LIN {X 0,Y 389.55,Z 544.012,A -85,B 0,C 180,E1 -11990.321,E2 -11990.321} C_VEL
LIN {X 0,Y 389.974,Z 535.473,A -85,B 0,C 180,E1 -11990.85,E2 -11990.85} C_VEL
LIN {X 0,Y 386.923,Z 515.614,A -85,B 0,C 180,E1 -11992.126,E2 -11992.126} C_VEL
LIN {X 0,Y 383.966,Z 500.348,A -85,B 0,C 180,E1 -11992.925,E2 -11992.925} C_VEL
LIN {X 0,Y 382.611,Z 493.228,A -85,B 0,C 180,E1 -11993.24,E2 -11993.24} C_VEL
LIN {X 0,Y 382.976,Z 485.45,A -85,B 0,C 180,E1 -11996.718,E2 -11996.718} C_VEL
LIN {X 0,Y 383.373,Z 478.936,A -85,B 0,C 180,E1 -11999.667,E2 -11999.667} C_VEL
LIN {X 0,Y 383.827,Z 471.033,A -85,B 0,C 180,E1 -12003.32,E2 -12003.32} C_VEL
LIN {X 0,Y 384.194,Z 464.514,A -85,B 0,C 180,E1 -12006.401,E2 -12006.401} C_VEL
LIN {X 0,Y 384.639,Z 457.344,A -85,B 0,C 180,E1 -12009.878,E2 -12009.878} C_VEL
LIN {X 0,Y 385.108,Z 450.851,A -85,B 0,C 180,E1 -12013.116,E2 -12013.116} C_VEL
LIN {X 0,Y 385.546,Z 444.924,A -85,B 0,C 180,E1 -12016.157,E2 -12016.157} C_VEL
LIN {X 0,Y 385.519,Z 440.793,A -85,B 0,C 180,E1 -12018.368,E2 -12018.368} C_VEL
LIN {X 0,Y 384.796,Z 436.258,A -85,B 0,C 180,E1 -12020.941,E2 -12020.941} C_VEL
LIN {X 0,Y 383.623,Z 429.852,A -85,B 0,C 180,E1 -12024.754,E2 -12024.754} C_VEL
LIN {X 0,Y 383.043,Z 426.398,A -85,B 0,C 180,E1 -12027.007,E2 -12027.007} C_VEL
LIN {X 0,Y 382.993,Z 426.406,A -85,B 0,C 180,E1 -12030.3,E2 -12030.3} C_VEL
LIN {X 0,Y 383.058,Z 426.39,A -85,B 0,C 180,E1 -12032.698,E2 -12032.698} C_VEL
LIN {X 0,Y 383.054,Z 426.391,A -85,B 0,C 180,E1 -12035.04,E2 -12035.04} C_VEL
LIN {X 0,Y 382.995,Z 426.395,A -85,B 0,C 180,E1 -12038.469,E2 -12038.469} C_VEL
LIN {X 0,Y 383.091,Z 426.391,A -85,B 0,C 180,E1 -12041.828,E2 -12041.828} C_VEL
LIN {X 0,Y 383.112,Z 426.374,A -85,B 0,C 180,E1 -12045.118,E2 -12045.118} C_VEL
LIN {X 0,Y 383.099,Z 426.39,A -85,B 0,C 180,E1 -12048.358,E2 -12048.358} C_VEL
LIN {X 0,Y 383.23,Z 426.363,A -85,B 0,C 180,E1 -12052.013,E2 -12052.013} C_VEL
LIN {X 0,Y 383.199,Z 426.376,A -85,B 0,C 180,E1 -12054.739,E2 -12054.739} C_VEL
LIN {X 0,Y 383.387,Z 426.343,A -85,B 0,C 180,E1 -12057.899,E2 -12057.899} C_VEL
LIN {X 0,Y 383.522,Z 426.34,A -85,B 0,C 180,E1 -12060,E2 -12060} C_VEL
LIN {X 0,Y 383.248,Z 426.358,A -85,B 0,C 180,E1 -12063.154,E2 -12063.154} C_VEL
LIN {X 0,Y 383.271,Z 426.365,A -85,B 0,C 180,E1 -12066.637,E2 -12066.637} C_VEL
LIN {X 0,Y 383.262,Z 426.356,A -85,B 0,C 180,E1 -12068.436,E2 -12068.436} C_VEL
LIN {X 0,Y 383.1,Z 426.391,A -85,B 0,C 180,E1 -12071.642,E2 -12071.642} C_VEL
LIN {X 0,Y 383.112,Z 426.383,A -85,B 0,C 180,E1 -12074.882,E2 -12074.882} C_VEL
LIN {X 0,Y 383.065,Z 426.386,A -85,B 0,C 180,E1 -12078.174,E2 -12078.174} C_VEL
LIN {X 0,Y 382.994,Z 426.402,A -85,B 0,C 180,E1 -12081.531,E2 -12081.531} C_VEL
LIN {X 0,Y 383.052,Z 426.396,A -85,B 0,C 180,E1 -12084.96,E2 -12084.96} C_VEL
LIN {X 0,Y 383.042,Z 426.4,A -85,B 0,C 180,E1 -12088.493,E2 -12088.493} C_VEL
LIN {X 0,Y 383.011,Z 426.401,A -85,B 0,C 180,E1 -12092.15,E2 -12092.15} C_VEL
LIN {X 0,Y 383.019,Z 426.401,A -85,B 0,C 180,E1 -12094.668,E2 -12094.668} C_VEL
LIN {X 0,Y 383.001,Z 426.401,A -85,B 0,C 180,E1 -12097.904,E2 -12097.904} C_VEL
LIN {X 0,Y 382.987,Z 426.405,A -85,B 0,C 180,E1 -12101.347,E2 -12101.347} C_VEL
LIN {X 0,Y 383.037,Z 426.473,A -85,B 0,C 180,E1 -12104.763,E2 -12104.763} C_VEL
LIN {X 0,Y 384.737,Z 434.782,A -85,B 0,C 180,E1 -12107.861,E2 -12107.861} C_VEL
LIN {X 0,Y 385.867,Z 441.672,A -85,B 0,C 180,E1 -12110.396,E2 -12110.396} C_VEL
LIN {X 0,Y 385.944,Z 445.456,A -85,B 0,C 180,E1 -12111.747,E2 -12111.747} C_VEL
LIN {X 0,Y 385.278,Z 456.469,A -85,B 0,C 180,E1 -12115.564,E2 -12115.564} C_VEL
LIN {X 0,Y 384.788,Z 467.116,A -85,B 0,C 180,E1 -12119.242,E2 -12119.242} C_VEL
LIN {X 0,Y 384.378,Z 475.927,A -85,B 0,C 180,E1 -12122.209,E2 -12122.209} C_VEL
LIN {X 0,Y 383.988,Z 486.577,A -85,B 0,C 180,E1 -12125.681,E2 -12125.681} C_VEL
LIN {X 0,Y 383.851,Z 491.515,A -85,B 0,C 180,E1 -12127.165,E2 -12127.165} C_VEL
LIN {X 0,Y 387.586,Z 506.42,A -85,B 0,C 180,E1 -12127.781,E2 -12127.781} C_VEL
LIN {X 0,Y 390.26,Z 520.477,A -85,B 0,C 180,E1 -12128.521,E2 -12128.521} C_VEL
LIN {X 0,Y 390.956,Z 526.338,A -85,B 0,C 180,E1 -12128.872,E2 -12128.872} C_VEL
LIN {X 0,Y 390.117,Z 538.424,A -85,B 0,C 180,E1 -12129.602,E2 -12129.602} C_VEL
LIN {X 0,Y 388.997,Z 551.518,A -85,B 0,C 180,E1 -12130.611,E2 -12130.611} C_VEL
LIN {X 0,Y 387.734,Z 563.629,A -85,B 0,C 180,E1 -12131.78,E2 -12131.78} C_VEL
LIN {X 0,Y 386.48,Z 574.62,A -85,B 0,C 180,E1 -12133.085,E2 -12133.085} C_VEL
LIN {X 0,Y 385.225,Z 585.417,A -85,B 0,C 180,E1 -12134.661,E2 -12134.661} C_VEL
LIN {X 0,Y 384.25,Z 594.334,A -85,B 0,C 180,E1 -12136.245,E2 -12136.245} C_VEL
LIN {X 0,Y 383.456,Z 601.761,A -85,B 0,C 180,E1 -12137.832,E2 -12137.832} C_VEL
LIN {X 0,Y 382.777,Z 607.952,A -85,B 0,C 180,E1 -12139.42,E2 -12139.42} C_VEL
LIN {X 0,Y 382.143,Z 614.494,A -85,B 0,C 180,E1 -12141.539,E2 -12141.539} C_VEL
LIN {X 0,Y 381.849,Z 619.404,A -85,B 0,C 180,E1 -12143.66,E2 -12143.66} C_VEL
LIN {X 0,Y 381.636,Z 622.825,A -85,B 0,C 180,E1 -12145.776,E2 -12145.776} C_VEL
LIN {X 0,Y 381.552,Z 624.859,A -85,B 0,C 180,E1 -12147.889,E2 -12147.889} C_VEL
LIN {X 0,Y 381.572,Z 625.56,A -85,B 0,C 180,E1 -12150,E2 -12150} C_VEL
LIN {X 0,Y 381.551,Z 624.928,A -85,B 0,C 180,E1 -12152.111,E2 -12152.111} C_VEL
LIN {X 0,Y 381.634,Z 622.952,A -85,B 0,C 180,E1 -12154.224,E2 -12154.224} C_VEL
LIN {X 0,Y 381.808,Z 619.592,A -85,B 0,C 180,E1 -12156.341,E2 -12156.341} C_VEL
LIN {X 0,Y 382.137,Z 614.75,A -85,B 0,C 180,E1 -12158.461,E2 -12158.461} C_VEL
LIN {X 0,Y 382.73,Z 608.275,A -85,B 0,C 180,E1 -12160.581,E2 -12160.581} C_VEL
LIN {X 0,Y 383.546,Z 601.057,A -85,B 0,C 180,E1 -12162.433,E2 -12162.433} C_VEL
LIN {X 0,Y 384.407,Z 592.904,A -85,B 0,C 180,E1 -12164.134,E2 -12164.134} C_VEL
LIN {X 0,Y 385.575,Z 582.661,A -85,B 0,C 180,E1 -12165.867,E2 -12165.867} C_VEL
LIN {X 0,Y 386.791,Z 572.244,A -85,B 0,C 180,E1 -12167.31,E2 -12167.31} C_VEL
LIN {X 0,Y 387.323,Z 567.013,A -85,B 0,C 180,E1 -12167.939,E2 -12167.939} C_VEL
LIN {X 0,Y 387.168,Z 562.405,A -85,B 0,C 180,E1 -12168.481,E2 -12168.481} C_VEL
LIN {X 0,Y 385.32,Z 554.726,A -85,B 0,C 180,E1 -12169.375,E2 -12169.375} C_VEL
LIN {X 0,Y 383.5,Z 546.778,A -85,B 0,C 180,E1 -12170.208,E2 -12170.208} C_VEL
LIN {X 0,Y 383.264,Z 541.619,A -85,B 0,C 180,E1 -12170.642,E2 -12170.642} C_VEL
LIN {X 0,Y 384.198,Z 529.103,A -85,B 0,C 180,E1 -12171.46,E2 -12171.46} C_VEL
LIN {X 0,Y 384.104,Z 524.85,A -85,B 0,C 180,E1 -12171.709,E2 -12171.709} C_VEL
LIN {X 0,Y 381.821,Z 511.485,A -85,B 0,C 180,E1 -12172.486,E2 -12172.486} C_VEL
LIN {X 0,Y 378.417,Z 497.286,A -85,B 0,C 180,E1 -12173.156,E2 -12173.156} C_VEL
LIN {X 0,Y 376.897,Z 491.19,A -85,B 0,C 180,E1 -12173.417,E2 -12173.417} C_VEL
LIN {X 0,Y 377.325,Z 479.65,A -85,B 0,C 180,E1 -12177.15,E2 -12177.15} C_VEL
LIN {X 0,Y 377.798,Z 469.278,A -85,B 0,C 180,E1 -12180.663,E2 -12180.663} C_VEL
LIN {X 0,Y 378.339,Z 458.238,A -85,B 0,C 180,E1 -12184.511,E2 -12184.511} C_VEL
LIN {X 0,Y 379.011,Z 447.434,A -85,B 0,C 180,E1 -12188.303,E2 -12188.303} C_VEL
LIN {X 0,Y 379.019,Z 443.422,A -85,B 0,C 180,E1 -12189.754,E2 -12189.754} C_VEL
LIN {X 0,Y 378.012,Z 437.363,A -85,B 0,C 180,E1 -12192.014,E2 -12192.014} C_VEL
LIN {X 0,Y 376.299,Z 428.906,A -85,B 0,C 180,E1 -12195.212,E2 -12195.212} C_VEL
LIN {X 0,Y 375.959,Z 427.284,A -85,B 0,C 180,E1 -12195.836,E2 -12195.836} C_VEL
LIN {X 0,Y 375.942,Z 427.289,A -85,B 0,C 180,E1 -12199.133,E2 -12199.133} C_VEL
LIN {X 0,Y 375.967,Z 427.283,A -85,B 0,C 180,E1 -12201.912,E2 -12201.912} C_VEL
LIN {X 0,Y 375.982,Z 427.273,A -85,B 0,C 180,E1 -12205.333,E2 -12205.333} C_VEL
LIN {X 0,Y 375.962,Z 427.279,A -85,B 0,C 180,E1 -12208.438,E2 -12208.438} C_VEL
LIN {X 0,Y 376.004,Z 427.274,A -85,B 0,C 180,E1 -12212.142,E2 -12212.142} C_VEL
LIN {X 0,Y 376.023,Z 427.359,A -85,B 0,C 180,E1 -12215.39,E2 -12215.39} C_VEL
LIN {X 0,Y 381.008,Z 442.581,A -85,B 0,C 180,E1 -12216.589,E2 -12216.589} C_VEL
LIN {X 0,Y 384.181,Z 453.208,A -85,B 0,C 180,E1 -12217.55,E2 -12217.55} C_VEL
LIN {X 0,Y 382.956,Z 467.291,A -85,B 0,C 180,E1 -12218.749,E2 -12218.749} C_VEL
LIN {X 0,Y 381.648,Z 480.803,A -85,B 0,C 180,E1 -12220.158,E2 -12220.158} C_VEL
LIN {X 0,Y 380.365,Z 492.989,A -85,B 0,C 180,E1 -12221.693,E2 -12221.693} C_VEL
LIN {X 0,Y 379.267,Z 503.692,A -85,B 0,C 180,E1 -12223.308,E2 -12223.308} C_VEL
LIN {X 0,Y 378.205,Z 512.753,A -85,B 0,C 180,E1 -12224.921,E2 -12224.921} C_VEL
LIN {X 0,Y 377.419,Z 521.639,A -85,B 0,C 180,E1 -12226.814,E2 -12226.814} C_VEL
LIN {X 0,Y 376.623,Z 529.015,A -85,B 0,C 180,E1 -12228.7,E2 -12228.7} C_VEL
LIN {X 0,Y 376.043,Z 535.823,A -85,B 0,C 180,E1 -12230.859,E2 -12230.859} C_VEL
LIN {X 0,Y 375.611,Z 540.995,A -85,B 0,C 180,E1 -12232.948,E2 -12232.948} C_VEL
LIN {X 0,Y 375.491,Z 544.234,A -85,B 0,C 180,E1 -12234.63,E2 -12234.63} C_VEL
LIN {X 0,Y 375.294,Z 547.209,A -85,B 0,C 180,E1 -12236.779,E2 -12236.779} C_VEL
LIN {X 0,Y 374.988,Z 548.983,A -85,B 0,C 180,E1 -12238.926,E2 -12238.926} C_VEL
LIN {X 0,Y 375.03,Z 549.543,A -85,B 0,C 180,E1 -12241.074,E2 -12241.074} C_VEL
LIN {X 0,Y 375.315,Z 548.902,A -85,B 0,C 180,E1 -12243.22,E2 -12243.22} C_VEL
LIN {X 0,Y 375.838,Z 547.056,A -85,B 0,C 180,E1 -12245.365,E2 -12245.365} C_VEL
LIN {X 0,Y 376.224,Z 544.012,A -85,B 0,C 180,E1 -12247.514,E2 -12247.514} C_VEL
LIN {X 0,Y 376.901,Z 539.622,A -85,B 0,C 180,E1 -12249.661,E2 -12249.661} C_VEL
LIN {X 0,Y 377.559,Z 533.837,A -85,B 0,C 180,E1 -12251.815,E2 -12251.815} C_VEL
LIN {X 0,Y 378.769,Z 526.39,A -85,B 0,C 180,E1 -12253.958,E2 -12253.958} C_VEL
LIN {X 0,Y 379.802,Z 519.659,A -85,B 0,C 180,E1 -12255.554,E2 -12255.554} C_VEL
LIN {X 0,Y 381.234,Z 510.121,A -85,B 0,C 180,E1 -12257.432,E2 -12257.432} C_VEL
LIN {X 0,Y 382.539,Z 500.397,A -85,B 0,C 180,E1 -12259.032,E2 -12259.032} C_VEL
LIN {X 0,Y 384.197,Z 488.421,A -85,B 0,C 180,E1 -12260.65,E2 -12260.65} C_VEL
LIN {X 0,Y 385.845,Z 475.738,A -85,B 0,C 180,E1 -12262.066,E2 -12262.066} C_VEL
LIN {X 0,Y 387.215,Z 462.86,A -85,B 0,C 180,E1 -12263.251,E2 -12263.251} C_VEL
LIN {X 0,Y 387.867,Z 456.283,A -85,B 0,C 180,E1 -12263.77,E2 -12263.77} C_VEL
LIN {X 0,Y 384.824,Z 446.725,A -85,B 0,C 180,E1 -12264.838,E2 -12264.838} C_VEL
LIN {X 0,Y 379.638,Z 434.754,A -85,B 0,C 180,E1 -12266.212,E2 -12266.212} C_VEL
LIN {X 0,Y 376.181,Z 428.125,A -85,B 0,C 180,E1 -12267.01,E2 -12267.01} C_VEL
LIN {X 0,Y 376.012,Z 427.277,A -85,B 0,C 180,E1 -12267.125,E2 -12267.125} C_VEL
LIN {X 0,Y 375.957,Z 427.28,A -85,B 0,C 180,E1 -12270.694,E2 -12270.694} C_VEL
LIN {X 0,Y 375.961,Z 427.28,A -85,B 0,C 180,E1 -12274.111,E2 -12274.111} C_VEL
LIN {X 0,Y 375.954,Z 427.281,A -85,B 0,C 180,E1 -12276.741,E2 -12276.741} C_VEL
LIN {X 0,Y 375.972,Z 427.343,A -85,B 0,C 180,E1 -12279.137,E2 -12279.137} C_VEL
LIN {X 0,Y 376.756,Z 431.554,A -85,B 0,C 180,E1 -12282.186,E2 -12282.186} C_VEL
LIN {X 0,Y 377.08,Z 434.855,A -85,B 0,C 180,E1 -12284.228,E2 -12284.228} C_VEL
LIN {X 0,Y 376.323,Z 441.536,A -85,B 0,C 180,E1 -12287.754,E2 -12287.754} C_VEL
LIN {X 0,Y 376.101,Z 448.65,A -85,B 0,C 180,E1 -12291.186,E2 -12291.186} C_VEL
LIN {X 0,Y 375.976,Z 456.213,A -85,B 0,C 180,E1 -12294.586,E2 -12294.586} C_VEL
LIN {X 0,Y 375.765,Z 465.202,A -85,B 0,C 180,E1 -12298.42,E2 -12298.42} C_VEL
LIN {X 0,Y 375.648,Z 472.795,A -85,B 0,C 180,E1 -12301.561,E2 -12301.561} C_VEL
LIN {X 0,Y 375.447,Z 480.867,A -85,B 0,C 180,E1 -12304.812,E2 -12304.812} C_VEL
LIN {X 0,Y 376.282,Z 484.869,A -85,B 0,C 180,E1 -12305.069,E2 -12305.069} C_VEL
LIN {X 0,Y 378.786,Z 495.627,A -85,B 0,C 180,E1 -12305.81,E2 -12305.81} C_VEL
LIN {X 0,Y 380.799,Z 508.736,A -85,B 0,C 180,E1 -12306.713,E2 -12306.713} C_VEL
LIN {X 0,Y 381.881,Z 525.377,A -85,B 0,C 180,E1 -12307.924,E2 -12307.924} C_VEL
LIN {X 0,Y 382.948,Z 534.73,A -85,B 0,C 180,E1 -12308.699,E2 -12308.699} C_VEL
LIN {X 0,Y 383.303,Z 538.44,A -85,B 0,C 180,E1 -12308.952,E2 -12308.952} C_VEL
LIN {X 0,Y 382.313,Z 551.26,A -85,B 0,C 180,E1 -12309.83,E2 -12309.83} C_VEL
LIN {X 0,Y 381.121,Z 563.56,A -85,B 0,C 180,E1 -12310.894,E2 -12310.894} C_VEL
LIN {X 0,Y 379.885,Z 574.724,A -85,B 0,C 180,E1 -12312.087,E2 -12312.087} C_VEL
LIN {X 0,Y 378.643,Z 585.901,A -85,B 0,C 180,E1 -12313.557,E2 -12313.557} C_VEL
LIN {X 0,Y 377.481,Z 595.928,A -85,B 0,C 180,E1 -12315.174,E2 -12315.174} C_VEL
LIN {X 0,Y 376.63,Z 604.166,A -85,B 0,C 180,E1 -12316.786,E2 -12316.786} C_VEL
LIN {X 0,Y 375.739,Z 612.057,A -85,B 0,C 180,E1 -12318.674,E2 -12318.674} C_VEL
LIN {X 0,Y 375.247,Z 617.578,A -85,B 0,C 180,E1 -12320.296,E2 -12320.296} C_VEL
LIN {X 0,Y 374.792,Z 623.348,A -85,B 0,C 180,E1 -12322.457,E2 -12322.457} C_VEL
LIN {X 0,Y 374.702,Z 626.071,A -85,B 0,C 180,E1 -12323.763,E2 -12323.763} C_VEL
LIN {X 0,Y 374.607,Z 629.077,A -85,B 0,C 180,E1 -12325.696,E2 -12325.696} C_VEL
LIN {X 0,Y 374.53,Z 631.117,A -85,B 0,C 180,E1 -12327.849,E2 -12327.849} C_VEL
LIN {X 0,Y 374.546,Z 631.796,A -85,B 0,C 180,E1 -12330,E2 -12330} C_VEL
LIN {X 0,Y 374.53,Z 631.117,A -85,B 0,C 180,E1 -12332.151,E2 -12332.151} C_VEL
LIN {X 0,Y 374.594,Z 629.077,A -85,B 0,C 180,E1 -12334.304,E2 -12334.304} C_VEL
LIN {X 0,Y 374.681,Z 625.627,A -85,B 0,C 180,E1 -12336.462,E2 -12336.462} C_VEL
LIN {X 0,Y 374.978,Z 620.661,A -85,B 0,C 180,E1 -12338.623,E2 -12338.623} C_VEL
LIN {X 0,Y 375.515,Z 614.034,A -85,B 0,C 180,E1 -12340.787,E2 -12340.787} C_VEL
LIN {X 0,Y 376.348,Z 606.612,A -85,B 0,C 180,E1 -12342.675,E2 -12342.675} C_VEL
LIN {X 0,Y 377.09,Z 598.979,A -85,B 0,C 180,E1 -12344.269,E2 -12344.269} C_VEL
LIN {X 0,Y 378.186,Z 589.435,A -85,B 0,C 180,E1 -12345.909,E2 -12345.909} C_VEL
LIN {X 0,Y 379.33,Z 578.998,A -85,B 0,C 180,E1 -12347.383,E2 -12347.383} C_VEL
LIN {X 0,Y 380.726,Z 567.452,A -85,B 0,C 180,E1 -12348.707,E2 -12348.707} C_VEL
LIN {X 0,Y 381.944,Z 555.302,A -85,B 0,C 180,E1 -12349.84,E2 -12349.84} C_VEL
LIN {X 0,Y 383.036,Z 541.993,A -85,B 0,C 180,E1 -12350.823,E2 -12350.823} C_VEL
LIN {X 0,Y 383.234,Z 536.565,A -85,B 0,C 180,E1 -12351.164,E2 -12351.164} C_VEL
LIN {X 0,Y 380.34,Z 517.81,A -85,B 0,C 180,E1 -12352.353,E2 -12352.353} C_VEL
LIN {X 0,Y 377.516,Z 502.717,A -85,B 0,C 180,E1 -12353.202,E2 -12353.202} C_VEL
LIN {X 0,Y 375.59,Z 492.591,A -85,B 0,C 180,E1 -12353.661,E2 -12353.661} C_VEL
LIN {X 0,Y 375.896,Z 486.003,A -85,B 0,C 180,E1 -12356.662,E2 -12356.662} C_VEL
LIN {X 0,Y 376.368,Z 478.188,A -85,B 0,C 180,E1 -12360.277,E2 -12360.277} C_VEL
LIN {X 0,Y 376.896,Z 470.272,A -85,B 0,C 180,E1 -12364.015,E2 -12364.015} C_VEL
LIN {X 0,Y 377.333,Z 462.216,A -85,B 0,C 180,E1 -12367.926,E2 -12367.926} C_VEL
LIN {X 0,Y 377.797,Z 455.488,A -85,B 0,C 180,E1 -12371.283,E2 -12371.283} C_VEL
LIN {X 0,Y 378.387,Z 448.045,A -85,B 0,C 180,E1 -12375.106,E2 -12375.106} C_VEL
LIN {X 0,Y 378.569,Z 442.74,A -85,B 0,C 180,E1 -12377.952,E2 -12377.952} C_VEL
LIN {X 0,Y 377.865,Z 437.777,A -85,B 0,C 180,E1 -12380.775,E2 -12380.775} C_VEL
LIN {X 0,Y 376.678,Z 431.324,A -85,B 0,C 180,E1 -12384.662,E2 -12384.662} C_VEL
LIN {X 0,Y 375.994,Z 427.276,A -85,B 0,C 180,E1 -12387.26,E2 -12387.26} C_VEL
LIN {X 0,Y 375.972,Z 427.28,A -85,B 0,C 180,E1 -12390.921,E2 -12390.921} C_VEL
LIN {X 0,Y 376.007,Z 427.262,A -85,B 0,C 180,E1 -12394.539,E2 -12394.539} C_VEL
LIN {X 0,Y 375.965,Z 427.274,A -85,B 0,C 180,E1 -12398.046,E2 -12398.046} C_VEL
LIN {X 0,Y 376.026,Z 427.269,A -85,B 0,C 180,E1 -12401.474,E2 -12401.474} C_VEL
LIN {X 0,Y 376.06,Z 427.253,A -85,B 0,C 180,E1 -12404.833,E2 -12404.833} C_VEL
LIN {X 0,Y 376.052,Z 427.269,A -85,B 0,C 180,E1 -12408.137,E2 -12408.137} C_VEL
LIN {X 0,Y 376.202,Z 427.238,A -85,B 0,C 180,E1 -12411.938,E2 -12411.938} C_VEL
LIN {X 0,Y 376.171,Z 427.252,A -85,B 0,C 180,E1 -12414.64,E2 -12414.64} C_VEL
LIN {X 0,Y 376.354,Z 427.219,A -85,B 0,C 180,E1 -12417.86,E2 -12417.86} C_VEL
LIN {X 0,Y 376.491,Z 427.216,A -85,B 0,C 180,E1 -12420,E2 -12420} C_VEL
LIN {X 0,Y 376.186,Z 427.237,A -85,B 0,C 180,E1 -12423.213,E2 -12423.213} C_VEL
LIN {X 0,Y 376.236,Z 427.241,A -85,B 0,C 180,E1 -12426.628,E2 -12426.628} C_VEL
LIN {X 0,Y 376.207,Z 427.235,A -85,B 0,C 180,E1 -12428.595,E2 -12428.595} C_VEL
LIN {X 0,Y 376.053,Z 427.269,A -85,B 0,C 180,E1 -12431.863,E2 -12431.863} C_VEL
LIN {X 0,Y 376.06,Z 427.264,A -85,B 0,C 180,E1 -12435.167,E2 -12435.167} C_VEL
LIN {X 0,Y 376.011,Z 427.263,A -85,B 0,C 180,E1 -12438.527,E2 -12438.527} C_VEL
LIN {X 0,Y 375.959,Z 427.278,A -85,B 0,C 180,E1 -12441.955,E2 -12441.955} C_VEL
LIN {X 0,Y 376.007,Z 427.273,A -85,B 0,C 180,E1 -12445.461,E2 -12445.461} C_VEL
LIN {X 0,Y 375.972,Z 427.277,A -85,B 0,C 180,E1 -12449.079,E2 -12449.079} C_VEL
LIN {X 0,Y 375.951,Z 427.278,A -85,B 0,C 180,E1 -12452.829,E2 -12452.829} C_VEL
LIN {X 0,Y 375.959,Z 427.276,A -85,B 0,C 180,E1 -12455.416,E2 -12455.416} C_VEL
LIN {X 0,Y 375.976,Z 427.277,A -85,B 0,C 180,E1 -12458.271,E2 -12458.271} C_VEL
LIN {X 0,Y 375.937,Z 427.283,A -85,B 0,C 180,E1 -12461.601,E2 -12461.601} C_VEL
LIN {X 0,Y 375.97,Z 427.294,A -85,B 0,C 180,E1 -12464.288,E2 -12464.288} C_VEL
LIN {X 0,Y 377.584,Z 435.211,A -85,B 0,C 180,E1 -12467.289,E2 -12467.289} C_VEL
LIN {X 0,Y 378.728,Z 441.181,A -85,B 0,C 180,E1 -12469.538,E2 -12469.538} C_VEL
LIN {X 0,Y 379.072,Z 445.563,A -85,B 0,C 180,E1 -12471.14,E2 -12471.14} C_VEL
LIN {X 0,Y 378.42,Z 456.099,A -85,B 0,C 180,E1 -12474.849,E2 -12474.849} C_VEL
LIN {X 0,Y 377.901,Z 466.875,A -85,B 0,C 180,E1 -12478.619,E2 -12478.619} C_VEL
LIN {X 0,Y 377.485,Z 475.778,A -85,B 0,C 180,E1 -12481.656,E2 -12481.656} C_VEL
LIN {X 0,Y 377.031,Z 486.532,A -85,B 0,C 180,E1 -12485.203,E2 -12485.203} C_VEL
LIN {X 0,Y 376.905,Z 491.373,A -85,B 0,C 180,E1 -12486.718,E2 -12486.718} C_VEL
LIN {X 0,Y 380.862,Z 507.204,A -85,B 0,C 180,E1 -12487.394,E2 -12487.394} C_VEL
LIN {X 0,Y 383.401,Z 520.5,A -85,B 0,C 180,E1 -12488.117,E2 -12488.117} C_VEL
LIN {X 0,Y 384.26,Z 527.394,A -85,B 0,C 180,E1 -12488.543,E2 -12488.543} C_VEL
LIN {X 0,Y 383.316,Z 540.363,A -85,B 0,C 180,E1 -12489.362,E2 -12489.362} C_VEL
LIN {X 0,Y 382.167,Z 553.079,A -85,B 0,C 180,E1 -12490.39,E2 -12490.39} C_VEL
LIN {X 0,Y 380.84,Z 564.864,A -85,B 0,C 180,E1 -12491.577,E2 -12491.577} C_VEL
LIN {X 0,Y 379.65,Z 574.673,A -85,B 0,C 180,E1 -12492.771,E2 -12492.771} C_VEL
LIN {X 0,Y 378.365,Z 585.472,A -85,B 0,C 180,E1 -12494.375,E2 -12494.375} C_VEL
LIN {X 0,Y 377.28,Z 594.392,A -85,B 0,C 180,E1 -12495.986,E2 -12495.986} C_VEL
LIN {X 0,Y 376.506,Z 601.819,A -85,B 0,C 180,E1 -12497.604,E2 -12497.604} C_VEL
LIN {X 0,Y 375.762,Z 608.011,A -85,B 0,C 180,E1 -12499.22,E2 -12499.22} C_VEL
LIN {X 0,Y 375.105,Z 614.553,A -85,B 0,C 180,E1 -12501.38,E2 -12501.38} C_VEL
LIN {X 0,Y 374.781,Z 619.463,A -85,B 0,C 180,E1 -12503.54,E2 -12503.54} C_VEL
LIN {X 0,Y 374.566,Z 622.884,A -85,B 0,C 180,E1 -12505.696,E2 -12505.696} C_VEL
LIN {X 0,Y 374.45,Z 624.918,A -85,B 0,C 180,E1 -12507.849,E2 -12507.849} C_VEL
LIN {X 0,Y 374.473,Z 625.618,A -85,B 0,C 180,E1 -12510,E2 -12510} C_VEL
LIN {X 0,Y 374.449,Z 624.987,A -85,B 0,C 180,E1 -12512.151,E2 -12512.151} C_VEL
LIN {X 0,Y 374.564,Z 623.009,A -85,B 0,C 180,E1 -12514.304,E2 -12514.304} C_VEL
LIN {X 0,Y 374.724,Z 619.649,A -85,B 0,C 180,E1 -12516.461,E2 -12516.461} C_VEL
LIN {X 0,Y 375.099,Z 614.807,A -85,B 0,C 180,E1 -12518.621,E2 -12518.621} C_VEL
LIN {X 0,Y 375.7,Z 608.33,A -85,B 0,C 180,E1 -12520.782,E2 -12520.782} C_VEL
LIN {X 0,Y 376.578,Z 601.11,A -85,B 0,C 180,E1 -12522.667,E2 -12522.667} C_VEL
LIN {X 0,Y 377.43,Z 593.474,A -85,B 0,C 180,E1 -12524.296,E2 -12524.296} C_VEL
LIN {X 0,Y 378.52,Z 584.438,A -85,B 0,C 180,E1 -12525.894,E2 -12525.894} C_VEL
LIN {X 0,Y 379.742,Z 574.381,A -85,B 0,C 180,E1 -12527.363,E2 -12527.363} C_VEL
LIN {X 0,Y 381.052,Z 563.308,A -85,B 0,C 180,E1 -12528.691,E2 -12528.691} C_VEL
LIN {X 0,Y 382.373,Z 551.107,A -85,B 0,C 180,E1 -12529.879,E2 -12529.879} C_VEL
LIN {X 0,Y 383.264,Z 541.619,A -85,B 0,C 180,E1 -12530.642,E2 -12530.642} C_VEL
LIN {X 0,Y 382.939,Z 538.171,A -85,B 0,C 180,E1 -12530.927,E2 -12530.927} C_VEL
LIN {X 0,Y 380.764,Z 532.824,A -85,B 0,C 180,E1 -12531.426,E2 -12531.426} C_VEL
LIN {X 0,Y 377.761,Z 526.324,A -85,B 0,C 180,E1 -12532.01,E2 -12532.01} C_VEL
LIN {X 0,Y 377.167,Z 523.952,A -85,B 0,C 180,E1 -12532.182,E2 -12532.182} C_VEL
LIN {X 0,Y 374.655,Z 510.038,A -85,B 0,C 180,E1 -12533.002,E2 -12533.002} C_VEL
LIN {X 0,Y 371.097,Z 495.685,A -85,B 0,C 180,E1 -12533.677,E2 -12533.677} C_VEL
LIN {X 0,Y 369.974,Z 491.187,A -85,B 0,C 180,E1 -12533.882,E2 -12533.882} C_VEL
LIN {X 0,Y 370.444,Z 479.532,A -85,B 0,C 180,E1 -12537.698,E2 -12537.698} C_VEL
LIN {X 0,Y 370.892,Z 469.493,A -85,B 0,C 180,E1 -12541.143,E2 -12541.143} C_VEL
LIN {X 0,Y 371.429,Z 459.685,A -85,B 0,C 180,E1 -12544.586,E2 -12544.586} C_VEL
LIN {X 0,Y 372.137,Z 448.564,A -85,B 0,C 180,E1 -12548.552,E2 -12548.552} C_VEL
LIN {X 0,Y 372.076,Z 444.723,A -85,B 0,C 180,E1 -12549.957,E2 -12549.957} C_VEL
LIN {X 0,Y 371.004,Z 438.405,A -85,B 0,C 180,E1 -12552.372,E2 -12552.372} C_VEL
LIN {X 0,Y 369.5,Z 430.888,A -85,B 0,C 180,E1 -12555.271,E2 -12555.271} C_VEL
LIN {X 0,Y 368.887,Z 428.163,A -85,B 0,C 180,E1 -12556.383,E2 -12556.383} C_VEL
LIN {X 0,Y 368.914,Z 428.164,A -85,B 0,C 180,E1 -12559.643,E2 -12559.643} C_VEL
LIN {X 0,Y 368.904,Z 428.155,A -85,B 0,C 180,E1 -12563.144,E2 -12563.144} C_VEL
LIN {X 0,Y 368.898,Z 428.152,A -85,B 0,C 180,E1 -12566.462,E2 -12566.462} C_VEL
LIN {X 0,Y 368.925,Z 428.148,A -85,B 0,C 180,E1 -12570.31,E2 -12570.31} C_VEL
LIN {X 0,Y 368.984,Z 428.149,A -85,B 0,C 180,E1 -12573.535,E2 -12573.535} C_VEL
LIN {X 0,Y 368.995,Z 428.147,A -85,B 0,C 180,E1 -12575.02,E2 -12575.02} C_VEL
LIN {X 0,Y 374.008,Z 443.613,A -85,B 0,C 180,E1 -12576.277,E2 -12576.277} C_VEL
LIN {X 0,Y 377.363,Z 454.655,A -85,B 0,C 180,E1 -12577.31,E2 -12577.31} C_VEL
LIN {X 0,Y 376.135,Z 468.173,A -85,B 0,C 180,E1 -12578.488,E2 -12578.488} C_VEL
LIN {X 0,Y 374.899,Z 480.239,A -85,B 0,C 180,E1 -12579.755,E2 -12579.755} C_VEL
LIN {X 0,Y 373.552,Z 492.85,A -85,B 0,C 180,E1 -12581.347,E2 -12581.347} C_VEL
LIN {X 0,Y 372.42,Z 503.706,A -85,B 0,C 180,E1 -12582.992,E2 -12582.992} C_VEL
LIN {X 0,Y 371.328,Z 512.897,A -85,B 0,C 180,E1 -12584.635,E2 -12584.635} C_VEL
LIN {X 0,Y 370.487,Z 521.903,A -85,B 0,C 180,E1 -12586.563,E2 -12586.563} C_VEL
LIN {X 0,Y 369.65,Z 529.386,A -85,B 0,C 180,E1 -12588.484,E2 -12588.484} C_VEL
LIN {X 0,Y 369.047,Z 536.294,A -85,B 0,C 180,E1 -12590.684,E2 -12590.684} C_VEL
LIN {X 0,Y 368.577,Z 541.712,A -85,B 0,C 180,E1 -12592.888,E2 -12592.888} C_VEL
LIN {X 0,Y 368.437,Z 544.843,A -85,B 0,C 180,E1 -12594.527,E2 -12594.527} C_VEL
LIN {X 0,Y 368.259,Z 547.891,A -85,B 0,C 180,E1 -12596.718,E2 -12596.718} C_VEL
LIN {X 0,Y 367.937,Z 549.734,A -85,B 0,C 180,E1 -12598.905,E2 -12598.905} C_VEL
LIN {X 0,Y 367.98,Z 550.366,A -85,B 0,C 180,E1 -12601.094,E2 -12601.094} C_VEL
LIN {X 0,Y 368.284,Z 549.794,A -85,B 0,C 180,E1 -12603.282,E2 -12603.282} C_VEL
LIN {X 0,Y 368.831,Z 548.008,A -85,B 0,C 180,E1 -12605.467,E2 -12605.467} C_VEL
LIN {X 0,Y 369.263,Z 545.022,A -85,B 0,C 180,E1 -12607.656,E2 -12607.656} C_VEL
LIN {X 0,Y 369.977,Z 540.725,A -85,B 0,C 180,E1 -12609.844,E2 -12609.844} C_VEL
LIN {X 0,Y 370.707,Z 535.011,A -85,B 0,C 180,E1 -12612.037,E2 -12612.037} C_VEL
LIN {X 0,Y 371.986,Z 527.63,A -85,B 0,C 180,E1 -12614.218,E2 -12614.218} C_VEL
LIN {X 0,Y 373.133,Z 520.824,A -85,B 0,C 180,E1 -12615.882,E2 -12615.882} C_VEL
LIN {X 0,Y 374.626,Z 511.579,A -85,B 0,C 180,E1 -12617.749,E2 -12617.749} C_VEL
LIN {X 0,Y 376.005,Z 501.988,A -85,B 0,C 180,E1 -12619.376,E2 -12619.376} C_VEL
LIN {X 0,Y 377.598,Z 491.263,A -85,B 0,C 180,E1 -12620.893,E2 -12620.893} C_VEL
LIN {X 0,Y 379.358,Z 478.98,A -85,B 0,C 180,E1 -12622.32,E2 -12622.32} C_VEL
LIN {X 0,Y 380.796,Z 466.751,A -85,B 0,C 180,E1 -12623.523,E2 -12623.523} C_VEL
LIN {X 0,Y 381.671,Z 459.206,A -85,B 0,C 180,E1 -12624.147,E2 -12624.147} C_VEL
LIN {X 0,Y 380.728,Z 455.019,A -85,B 0,C 180,E1 -12624.615,E2 -12624.615} C_VEL
LIN {X 0,Y 376.706,Z 444.132,A -85,B 0,C 180,E1 -12625.927,E2 -12625.927} C_VEL
LIN {X 0,Y 370.633,Z 431.883,A -85,B 0,C 180,E1 -12627.497,E2 -12627.497} C_VEL
LIN {X 0,Y 369.191,Z 429.255,A -85,B 0,C 180,E1 -12627.847,E2 -12627.847} C_VEL
LIN {X 0,Y 368.968,Z 428.155,A -85,B 0,C 180,E1 -12627.97,E2 -12627.97} C_VEL
LIN {X 0,Y 368.911,Z 428.158,A -85,B 0,C 180,E1 -12630.987,E2 -12630.987} C_VEL
LIN {X 0,Y 368.937,Z 428.155,A -85,B 0,C 180,E1 -12634.853,E2 -12634.853} C_VEL
LIN {X 0,Y 368.949,Z 428.336,A -85,B 0,C 180,E1 -12638.648,E2 -12638.648} C_VEL
LIN {X 0,Y 369.71,Z 432.333,A -85,B 0,C 180,E1 -12641.708,E2 -12641.708} C_VEL
LIN {X 0,Y 370.099,Z 435.56,A -85,B 0,C 180,E1 -12643.813,E2 -12643.813} C_VEL
LIN {X 0,Y 369.586,Z 439.934,A -85,B 0,C 180,E1 -12646.27,E2 -12646.27} C_VEL
LIN {X 0,Y 369.12,Z 447.978,A -85,B 0,C 180,E1 -12650.369,E2 -12650.369} C_VEL
LIN {X 0,Y 368.97,Z 455.315,A -85,B 0,C 180,E1 -12653.809,E2 -12653.809} C_VEL
LIN {X 0,Y 368.773,Z 462.48,A -85,B 0,C 180,E1 -12656.987,E2 -12656.987} C_VEL
LIN {X 0,Y 368.625,Z 471.492,A -85,B 0,C 180,E1 -12660.84,E2 -12660.84} C_VEL
LIN {X 0,Y 368.391,Z 478.966,A -85,B 0,C 180,E1 -12663.953,E2 -12663.953} C_VEL
LIN {X 0,Y 369.157,Z 482.836,A -85,B 0,C 180,E1 -12664.219,E2 -12664.219} C_VEL
LIN {X 0,Y 369.913,Z 485.255,A -85,B 0,C 180,E1 -12664.416,E2 -12664.416} C_VEL
LIN {X 0,Y 372.772,Z 498.1,A -85,B 0,C 180,E1 -12665.377,E2 -12665.377} C_VEL
LIN {X 0,Y 374.515,Z 510.44,A -85,B 0,C 180,E1 -12666.291,E2 -12666.291} C_VEL
LIN {X 0,Y 375.305,Z 526.086,A -85,B 0,C 180,E1 -12667.509,E2 -12667.509} C_VEL
LIN {X 0,Y 376.255,Z 535.945,A -85,B 0,C 180,E1 -12668.381,E2 -12668.381} C_VEL
LIN {X 0,Y 376.602,Z 539.654,A -85,B 0,C 180,E1 -12668.638,E2 -12668.638} C_VEL
LIN {X 0,Y 375.479,Z 553.01,A -85,B 0,C 180,E1 -12669.595,E2 -12669.595} C_VEL
LIN {X 0,Y 374.263,Z 564.87,A -85,B 0,C 180,E1 -12670.673,E2 -12670.673} C_VEL
LIN {X 0,Y 372.858,Z 576.849,A -85,B 0,C 180,E1 -12672.022,E2 -12672.022} C_VEL
LIN {X 0,Y 371.592,Z 587.631,A -85,B 0,C 180,E1 -12673.519,E2 -12673.519} C_VEL
LIN {X 0,Y 370.419,Z 597.327,A -85,B 0,C 180,E1 -12675.16,E2 -12675.16} C_VEL
LIN {X 0,Y 369.53,Z 605.343,A -85,B 0,C 180,E1 -12676.807,E2 -12676.807} C_VEL
LIN {X 0,Y 368.723,Z 612.002,A -85,B 0,C 180,E1 -12678.455,E2 -12678.455} C_VEL
LIN {X 0,Y 368.199,Z 617.522,A -85,B 0,C 180,E1 -12680.108,E2 -12680.108} C_VEL
LIN {X 0,Y 367.829,Z 622.036,A -85,B 0,C 180,E1 -12681.761,E2 -12681.761} C_VEL
LIN {X 0,Y 367.593,Z 626.346,A -85,B 0,C 180,E1 -12683.82,E2 -12683.82} C_VEL
LIN {X 0,Y 367.51,Z 629.019,A -85,B 0,C 180,E1 -12685.613,E2 -12685.613} C_VEL
LIN {X 0,Y 367.427,Z 631.059,A -85,B 0,C 180,E1 -12687.808,E2 -12687.808} C_VEL
LIN {X 0,Y 367.446,Z 631.738,A -85,B 0,C 180,E1 -12690,E2 -12690} C_VEL
LIN {X 0,Y 367.427,Z 631.058,A -85,B 0,C 180,E1 -12692.192,E2 -12692.192} C_VEL
LIN {X 0,Y 367.496,Z 629.018,A -85,B 0,C 180,E1 -12694.387,E2 -12694.387} C_VEL
LIN {X 0,Y 367.595,Z 625.568,A -85,B 0,C 180,E1 -12696.587,E2 -12696.587} C_VEL
LIN {X 0,Y 367.944,Z 620.603,A -85,B 0,C 180,E1 -12698.79,E2 -12698.79} C_VEL
LIN {X 0,Y 368.495,Z 613.976,A -85,B 0,C 180,E1 -12700.995,E2 -12700.995} C_VEL
LIN {X 0,Y 369.382,Z 606.555,A -85,B 0,C 180,E1 -12702.918,E2 -12702.918} C_VEL
LIN {X 0,Y 370.161,Z 598.923,A -85,B 0,C 180,E1 -12704.542,E2 -12704.542} C_VEL
LIN {X 0,Y 371.341,Z 589.381,A -85,B 0,C 180,E1 -12706.21,E2 -12706.21} C_VEL
LIN {X 0,Y 372.555,Z 578.946,A -85,B 0,C 180,E1 -12707.709,E2 -12707.709} C_VEL
LIN {X 0,Y 373.993,Z 567.403,A -85,B 0,C 180,E1 -12709.057,E2 -12709.057} C_VEL
LIN {X 0,Y 375.302,Z 554.7,A -85,B 0,C 180,E1 -12710.257,E2 -12710.257} C_VEL
LIN {X 0,Y 376.392,Z 541.947,A -85,B 0,C 180,E1 -12711.209,E2 -12711.209} C_VEL
LIN {X 0,Y 376.509,Z 537.649,A -85,B 0,C 180,E1 -12711.489,E2 -12711.489} C_VEL
LIN {X 0,Y 374.588,Z 524.889,A -85,B 0,C 180,E1 -12712.324,E2 -12712.324} C_VEL
LIN {X 0,Y 370.506,Z 502.226,A -85,B 0,C 180,E1 -12713.618,E2 -12713.618} C_VEL
LIN {X 0,Y 368.538,Z 491.907,A -85,B 0,C 180,E1 -12714.106,E2 -12714.106} C_VEL
LIN {X 0,Y 368.867,Z 485.24,A -85,B 0,C 180,E1 -12717.211,E2 -12717.211} C_VEL
LIN {X 0,Y 369.296,Z 478.733,A -85,B 0,C 180,E1 -12720.286,E2 -12720.286} C_VEL
LIN {X 0,Y 369.831,Z 470.814,A -85,B 0,C 180,E1 -12724.097,E2 -12724.097} C_VEL
LIN {X 0,Y 370.313,Z 462.747,A -85,B 0,C 180,E1 -12728.083,E2 -12728.083} C_VEL
LIN {X 0,Y 370.804,Z 455.911,A -85,B 0,C 180,E1 -12731.557,E2 -12731.557} C_VEL
LIN {X 0,Y 371.341,Z 449.292,A -85,B 0,C 180,E1 -12735.011,E2 -12735.011} C_VEL
LIN {X 0,Y 371.587,Z 444.664,A -85,B 0,C 180,E1 -12737.53,E2 -12737.53} C_VEL
LIN {X 0,Y 371.129,Z 440.461,A -85,B 0,C 180,E1 -12739.92,E2 -12739.92} C_VEL
LIN {X 0,Y 370.219,Z 435.542,A -85,B 0,C 180,E1 -12742.873,E2 -12742.873} C_VEL
LIN {X 0,Y 369.118,Z 429.112,A -85,B 0,C 180,E1 -12746.904,E2 -12746.904} C_VEL
LIN {X 0,Y 368.926,Z 428.157,A -85,B 0,C 180,E1 -12747.546,E2 -12747.546} C_VEL
LIN {X 0,Y 368.981,Z 428.15,A -85,B 0,C 180,E1 -12751.564,E2 -12751.564} C_VEL
LIN {X 0,Y 369.001,Z 428.132,A -85,B 0,C 180,E1 -12754.02,E2 -12754.02} C_VEL
LIN {X 0,Y 368.934,Z 428.151,A -85,B 0,C 180,E1 -12757.605,E2 -12757.605} C_VEL
LIN {X 0,Y 368.984,Z 428.146,A -85,B 0,C 180,E1 -12761.107,E2 -12761.107} C_VEL
LIN {X 0,Y 368.999,Z 428.134,A -85,B 0,C 180,E1 -12764.535,E2 -12764.535} C_VEL
LIN {X 0,Y 369.007,Z 428.147,A -85,B 0,C 180,E1 -12767.907,E2 -12767.907} C_VEL
LIN {X 0,Y 369.149,Z 428.116,A -85,B 0,C 180,E1 -12771.889,E2 -12771.889} C_VEL
LIN {X 0,Y 369.143,Z 428.128,A -85,B 0,C 180,E1 -12774.538,E2 -12774.538} C_VEL
LIN {X 0,Y 369.319,Z 428.095,A -85,B 0,C 180,E1 -12777.819,E2 -12777.819} C_VEL
LIN {X 0,Y 369.46,Z 428.091,A -85,B 0,C 180,E1 -12780,E2 -12780} C_VEL
LIN {X 0,Y 369.318,Z 428.096,A -85,B 0,C 180,E1 -12782.181,E2 -12782.181} C_VEL
LIN {X 0,Y 369.206,Z 428.118,A -85,B 0,C 180,E1 -12786.615,E2 -12786.615} C_VEL
LIN {X 0,Y 369.139,Z 428.115,A -85,B 0,C 180,E1 -12788.761,E2 -12788.761} C_VEL
LIN {X 0,Y 369.008,Z 428.144,A -85,B 0,C 180,E1 -12792.093,E2 -12792.093} C_VEL
LIN {X 0,Y 369,Z 428.147,A -85,B 0,C 180,E1 -12795.465,E2 -12795.465} C_VEL
LIN {X 0,Y 368.96,Z 428.141,A -85,B 0,C 180,E1 -12798.894,E2 -12798.894} C_VEL
LIN {X 0,Y 368.926,Z 428.149,A -85,B 0,C 180,E1 -12802.396,E2 -12802.396} C_VEL
LIN {X 0,Y 369.001,Z 428.142,A -85,B 0,C 180,E1 -12805.98,E2 -12805.98} C_VEL
LIN {X 0,Y 368.963,Z 428.151,A -85,B 0,C 180,E1 -12808.812,E2 -12808.812} C_VEL
LIN {X 0,Y 368.9,Z 428.158,A -85,B 0,C 180,E1 -12812.238,E2 -12812.238} C_VEL
LIN {X 0,Y 368.93,Z 428.154,A -85,B 0,C 180,E1 -12815.002,E2 -12815.002} C_VEL
LIN {X 0,Y 368.911,Z 428.159,A -85,B 0,C 180,E1 -12818.64,E2 -12818.64} C_VEL
LIN {X 0,Y 368.883,Z 428.163,A -85,B 0,C 180,E1 -12822.01,E2 -12822.01} C_VEL
LIN {X 0,Y 368.931,Z 428.292,A -85,B 0,C 180,E1 -12823.843,E2 -12823.843} C_VEL
LIN {X 0,Y 370.584,Z 436.288,A -85,B 0,C 180,E1 -12826.943,E2 -12826.943} C_VEL
LIN {X 0,Y 371.91,Z 443.229,A -85,B 0,C 180,E1 -12829.596,E2 -12829.596} C_VEL
LIN {X 0,Y 372.162,Z 448.257,A -85,B 0,C 180,E1 -12831.451,E2 -12831.451} C_VEL
LIN {X 0,Y 371.428,Z 459.4,A -85,B 0,C 180,E1 -12835.414,E2 -12835.414} C_VEL
LIN {X 0,Y 370.905,Z 470.242,A -85,B 0,C 180,E1 -12839.229,E2 -12839.229} C_VEL
LIN {X 0,Y 370.448,Z 479.225,A -85,B 0,C 180,E1 -12842.302,E2 -12842.302} C_VEL
LIN {X 0,Y 369.992,Z 491.399,A -85,B 0,C 180,E1 -12846.258,E2 -12846.258} C_VEL
LIN {X 0,Y 373.906,Z 506.919,A -85,B 0,C 180,E1 -12846.939,E2 -12846.939} C_VEL
LIN {X 0,Y 376.625,Z 520.589,A -85,B 0,C 180,E1 -12847.705,E2 -12847.705} C_VEL
LIN {X 0,Y 377.58,Z 528.532,A -85,B 0,C 180,E1 -12848.209,E2 -12848.209} C_VEL
LIN {X 0,Y 376.551,Z 542.04,A -85,B 0,C 180,E1 -12849.104,E2 -12849.104} C_VEL
LIN {X 0,Y 375.329,Z 554.521,A -85,B 0,C 180,E1 -12850.16,E2 -12850.16} C_VEL
LIN {X 0,Y 373.894,Z 566.064,A -85,B 0,C 180,E1 -12851.365,E2 -12851.365} C_VEL
LIN {X 0,Y 372.637,Z 576.645,A -85,B 0,C 180,E1 -12852.72,E2 -12852.72} C_VEL
LIN {X 0,Y 371.305,Z 587.126,A -85,B 0,C 180,E1 -12854.352,E2 -12854.352} C_VEL
LIN {X 0,Y 370.321,Z 594.449,A -85,B 0,C 180,E1 -12855.717,E2 -12855.717} C_VEL
LIN {X 0,Y 369.556,Z 601.877,A -85,B 0,C 180,E1 -12857.367,E2 -12857.367} C_VEL
LIN {X 0,Y 368.733,Z 608.069,A -85,B 0,C 180,E1 -12859.012,E2 -12859.012} C_VEL
LIN {X 0,Y 368.055,Z 614.612,A -85,B 0,C 180,E1 -12861.213,E2 -12861.213} C_VEL
LIN {X 0,Y 367.695,Z 619.522,A -85,B 0,C 180,E1 -12863.415,E2 -12863.415} C_VEL
LIN {X 0,Y 367.475,Z 622.943,A -85,B 0,C 180,E1 -12865.613,E2 -12865.613} C_VEL
LIN {X 0,Y 367.352,Z 624.977,A -85,B 0,C 180,E1 -12867.807,E2 -12867.807} C_VEL
LIN {X 0,Y 367.373,Z 625.677,A -85,B 0,C 180,E1 -12870,E2 -12870} C_VEL
LIN {X 0,Y 367.351,Z 625.045,A -85,B 0,C 180,E1 -12872.193,E2 -12872.193} C_VEL
LIN {X 0,Y 367.473,Z 623.067,A -85,B 0,C 180,E1 -12874.387,E2 -12874.387} C_VEL
LIN {X 0,Y 367.647,Z 619.706,A -85,B 0,C 180,E1 -12876.586,E2 -12876.586} C_VEL
LIN {X 0,Y 368.048,Z 614.863,A -85,B 0,C 180,E1 -12878.787,E2 -12878.787} C_VEL
LIN {X 0,Y 368.503,Z 610.169,A -85,B 0,C 180,E1 -12880.439,E2 -12880.439} C_VEL
LIN {X 0,Y 369.346,Z 603.363,A -85,B 0,C 180,E1 -12882.361,E2 -12882.361} C_VEL
LIN {X 0,Y 370.205,Z 596.25,A -85,B 0,C 180,E1 -12884.007,E2 -12884.007} C_VEL
LIN {X 0,Y 371.268,Z 587.688,A -85,B 0,C 180,E1 -12885.649,E2 -12885.649} C_VEL
LIN {X 0,Y 372.563,Z 577.317,A -85,B 0,C 180,E1 -12887.284,E2 -12887.284} C_VEL
LIN {X 0,Y 374.008,Z 565.718,A -85,B 0,C 180,E1 -12888.772,E2 -12888.772} C_VEL
LIN {X 0,Y 375.374,Z 554.097,A -85,B 0,C 180,E1 -12889.98,E2 -12889.98} C_VEL
LIN {X 0,Y 376.617,Z 541.651,A -85,B 0,C 180,E1 -12891.025,E2 -12891.025} C_VEL
LIN {X 0,Y 377.646,Z 527.781,A -85,B 0,C 180,E1 -12891.932,E2 -12891.932} C_VEL
LIN {X 0,Y 377.167,Z 523.952,A -85,B 0,C 180,E1 -12892.182,E2 -12892.182} C_VEL
LIN {X 0,Y 375.653,Z 518.798,A -85,B 0,C 180,E1 -12892.557,E2 -12892.557} C_VEL
LIN {X 0,Y 371.309,Z 510.894,A -85,B 0,C 180,E1 -12893.194,E2 -12893.194} C_VEL
LIN {X 0,Y 366.698,Z 502.905,A -85,B 0,C 180,E1 -12893.783,E2 -12893.783} C_VEL
LIN {X 0,Y 364.72,Z 497.606,A -85,B 0,C 180,E1 -12894.067,E2 -12894.067} C_VEL
LIN {X 0,Y 363.033,Z 491.182,A -85,B 0,C 180,E1 -12894.368,E2 -12894.368} C_VEL
LIN {X 0,Y 363.47,Z 481.27,A -85,B 0,C 180,E1 -12897.649,E2 -12897.649} C_VEL
LIN {X 0,Y 363.938,Z 472.157,A -85,B 0,C 180,E1 -12900.78,E2 -12900.78} C_VEL
LIN {X 0,Y 364.523,Z 461.203,A -85,B 0,C 180,E1 -12904.664,E2 -12904.664} C_VEL
LIN {X 0,Y 365.268,Z 450.024,A -85,B 0,C 180,E1 -12908.706,E2 -12908.706} C_VEL
LIN {X 0,Y 365.167,Z 445.985,A -85,B 0,C 180,E1 -12910.207,E2 -12910.207} C_VEL
LIN {X 0,Y 363.984,Z 439.297,A -85,B 0,C 180,E1 -12912.8,E2 -12912.8} C_VEL
LIN {X 0,Y 362.414,Z 431.522,A -85,B 0,C 180,E1 -12915.849,E2 -12915.849} C_VEL
LIN {X 0,Y 361.843,Z 429.043,A -85,B 0,C 180,E1 -12916.91,E2 -12916.91} C_VEL
LIN {X 0,Y 361.857,Z 429.039,A -85,B 0,C 180,E1 -12920.139,E2 -12920.139} C_VEL
LIN {X 0,Y 361.87,Z 429.031,A -85,B 0,C 180,E1 -12922.982,E2 -12922.982} C_VEL
LIN {X 0,Y 361.86,Z 429.029,A -85,B 0,C 180,E1 -12926.63,E2 -12926.63} C_VEL
LIN {X 0,Y 361.878,Z 429.022,A -85,B 0,C 180,E1 -12929.672,E2 -12929.672} C_VEL
LIN {X 0,Y 361.957,Z 429.024,A -85,B 0,C 180,E1 -12933.475,E2 -12933.475} C_VEL
LIN {X 0,Y 361.937,Z 429.025,A -85,B 0,C 180,E1 -12934.672,E2 -12934.672} C_VEL
LIN {X 0,Y 366.535,Z 443.053,A -85,B 0,C 180,E1 -12935.821,E2 -12935.821} C_VEL
LIN {X 0,Y 370.358,Z 455.4,A -85,B 0,C 180,E1 -12936.992,E2 -12936.992} C_VEL
LIN {X 0,Y 369.994,Z 461.948,A -85,B 0,C 180,E1 -12937.555,E2 -12937.555} C_VEL
LIN {X 0,Y 368.617,Z 475.572,A -85,B 0,C 180,E1 -12938.886,E2 -12938.886} C_VEL
LIN {X 0,Y 367.235,Z 488.586,A -85,B 0,C 180,E1 -12940.433,E2 -12940.433} C_VEL
LIN {X 0,Y 365.956,Z 500.266,A -85,B 0,C 180,E1 -12942.105,E2 -12942.105} C_VEL
LIN {X 0,Y 364.821,Z 510.092,A -85,B 0,C 180,E1 -12943.78,E2 -12943.78} C_VEL
LIN {X 0,Y 363.875,Z 518.449,A -85,B 0,C 180,E1 -12945.458,E2 -12945.458} C_VEL
LIN {X 0,Y 362.985,Z 526.656,A -85,B 0,C 180,E1 -12947.419,E2 -12947.419} C_VEL
LIN {X 0,Y 362.318,Z 533.448,A -85,B 0,C 180,E1 -12949.381,E2 -12949.381} C_VEL
LIN {X 0,Y 361.759,Z 539.671,A -85,B 0,C 180,E1 -12951.622,E2 -12951.622} C_VEL
LIN {X 0,Y 361.38,Z 544.457,A -85,B 0,C 180,E1 -12953.86,E2 -12953.86} C_VEL
LIN {X 0,Y 361.325,Z 547.144,A -85,B 0,C 180,E1 -12955.538,E2 -12955.538} C_VEL
LIN {X 0,Y 361.01,Z 549.672,A -85,B 0,C 180,E1 -12957.769,E2 -12957.769} C_VEL
LIN {X 0,Y 360.878,Z 550.989,A -85,B 0,C 180,E1 -12960,E2 -12960} C_VEL
LIN {X 0,Y 361.059,Z 551.093,A -85,B 0,C 180,E1 -12962.231,E2 -12962.231} C_VEL
LIN {X 0,Y 361.554,Z 549.981,A -85,B 0,C 180,E1 -12964.459,E2 -12964.459} C_VEL
LIN {X 0,Y 361.968,Z 547.699,A -85,B 0,C 180,E1 -12966.69,E2 -12966.69} C_VEL
LIN {X 0,Y 362.644,Z 544.136,A -85,B 0,C 180,E1 -12968.919,E2 -12968.919} C_VEL
LIN {X 0,Y 363.464,Z 539.2,A -85,B 0,C 180,E1 -12971.149,E2 -12971.149} C_VEL
LIN {X 0,Y 364.202,Z 534.54,A -85,B 0,C 180,E1 -12972.821,E2 -12972.821} C_VEL
LIN {X 0,Y 365.402,Z 527.921,A -85,B 0,C 180,E1 -12974.764,E2 -12974.764} C_VEL
LIN {X 0,Y 366.669,Z 520.906,A -85,B 0,C 180,E1 -12976.466,E2 -12976.466} C_VEL
LIN {X 0,Y 368.262,Z 511.626,A -85,B 0,C 180,E1 -12978.354,E2 -12978.354} C_VEL
LIN {X 0,Y 369.838,Z 501.877,A -85,B 0,C 180,E1 -12980.002,E2 -12980.002} C_VEL
LIN {X 0,Y 371.721,Z 489.749,A -85,B 0,C 180,E1 -12981.702,E2 -12981.702} C_VEL
LIN {X 0,Y 373.565,Z 477.358,A -85,B 0,C 180,E1 -12983.124,E2 -12983.124} C_VEL
LIN {X 0,Y 375.318,Z 463.305,A -85,B 0,C 180,E1 -12984.455,E2 -12984.455} C_VEL
LIN {X 0,Y 375.375,Z 459.945,A -85,B 0,C 180,E1 -12984.764,E2 -12984.764} C_VEL
LIN {X 0,Y 371.779,Z 449.338,A -85,B 0,C 180,E1 -12986.112,E2 -12986.112} C_VEL
LIN {X 0,Y 366.412,Z 437.765,A -85,B 0,C 180,E1 -12987.685,E2 -12987.685} C_VEL
LIN {X 0,Y 362.127,Z 430.076,A -85,B 0,C 180,E1 -12988.816,E2 -12988.816} C_VEL
LIN {X 0,Y 361.926,Z 429.031,A -85,B 0,C 180,E1 -12988.932,E2 -12988.932} C_VEL
LIN {X 0,Y 361.849,Z 429.038,A -85,B 0,C 180,E1 -12992.945,E2 -12992.945} C_VEL
LIN {X 0,Y 361.869,Z 429.036,A -85,B 0,C 180,E1 -12995.637,E2 -12995.637} C_VEL
LIN {X 0,Y 361.882,Z 429.123,A -85,B 0,C 180,E1 -12997.933,E2 -12997.933} C_VEL
LIN {X 0,Y 362.623,Z 433.165,A -85,B 0,C 180,E1 -13001.22,E2 -13001.22} C_VEL
LIN {X 0,Y 363.097,Z 436.33,A -85,B 0,C 180,E1 -13003.403,E2 -13003.403} C_VEL
LIN {X 0,Y 362.925,Z 439.018,A -85,B 0,C 180,E1 -13005.023,E2 -13005.023} C_VEL
LIN {X 0,Y 362.218,Z 446.69,A -85,B 0,C 180,E1 -13009.174,E2 -13009.174} C_VEL
LIN {X 0,Y 361.942,Z 454.464,A -85,B 0,C 180,E1 -13012.991,E2 -13012.991} C_VEL
LIN {X 0,Y 361.757,Z 461.506,A -85,B 0,C 180,E1 -13016.236,E2 -13016.236} C_VEL
LIN {X 0,Y 361.502,Z 469.202,A -85,B 0,C 180,E1 -13019.637,E2 -13019.637} C_VEL
LIN {X 0,Y 361.42,Z 475.093,A -85,B 0,C 180,E1 -13022.18,E2 -13022.18} C_VEL
LIN {X 0,Y 361.39,Z 476.997,A -85,B 0,C 180,E1 -13022.995,E2 -13022.995} C_VEL
LIN {X 0,Y 362.206,Z 481.102,A -85,B 0,C 180,E1 -13023.314,E2 -13023.314} C_VEL
LIN {X 0,Y 362.942,Z 483.295,A -85,B 0,C 180,E1 -13023.518,E2 -13023.518} C_VEL
LIN {X 0,Y 365.891,Z 495.497,A -85,B 0,C 180,E1 -13024.525,E2 -13024.525} C_VEL
LIN {X 0,Y 367.995,Z 509.479,A -85,B 0,C 180,E1 -13025.64,E2 -13025.64} C_VEL
LIN {X 0,Y 368.754,Z 524.46,A -85,B 0,C 180,E1 -13026.864,E2 -13026.864} C_VEL
LIN {X 0,Y 369.24,Z 534.243,A -85,B 0,C 180,E1 -13027.772,E2 -13027.772} C_VEL
LIN {X 0,Y 369.96,Z 539.968,A -85,B 0,C 180,E1 -13028.258,E2 -13028.258} C_VEL
LIN {X 0,Y 368.798,Z 553.08,A -85,B 0,C 180,E1 -13029.218,E2 -13029.218} C_VEL
LIN {X 0,Y 367.535,Z 564.829,A -85,B 0,C 180,E1 -13030.304,E2 -13030.304} C_VEL
LIN {X 0,Y 366.087,Z 576.803,A -85,B 0,C 180,E1 -13031.678,E2 -13031.678} C_VEL
LIN {X 0,Y 364.739,Z 587.582,A -85,B 0,C 180,E1 -13033.2,E2 -13033.2} C_VEL
LIN {X 0,Y 363.51,Z 597.275,A -85,B 0,C 180,E1 -13034.871,E2 -13034.871} C_VEL
LIN {X 0,Y 362.558,Z 605.289,A -85,B 0,C 180,E1 -13036.549,E2 -13036.549} C_VEL
LIN {X 0,Y 361.739,Z 611.947,A -85,B 0,C 180,E1 -13038.229,E2 -13038.229} C_VEL
LIN {X 0,Y 361.168,Z 617.466,A -85,B 0,C 180,E1 -13039.914,E2 -13039.914} C_VEL
LIN {X 0,Y 360.663,Z 623.234,A -85,B 0,C 180,E1 -13042.16,E2 -13042.16} C_VEL
LIN {X 0,Y 360.446,Z 627.419,A -85,B 0,C 180,E1 -13044.405,E2 -13044.405} C_VEL
LIN {X 0,Y 360.337,Z 630.152,A -85,B 0,C 180,E1 -13046.646,E2 -13046.646} C_VEL
LIN {X 0,Y 360.344,Z 631.51,A -85,B 0,C 180,E1 -13048.882,E2 -13048.882} C_VEL
LIN {X 0,Y 360.344,Z 631.509,A -85,B 0,C 180,E1 -13051.118,E2 -13051.118} C_VEL
LIN {X 0,Y 360.335,Z 630.151,A -85,B 0,C 180,E1 -13053.354,E2 -13053.354} C_VEL
LIN {X 0,Y 360.413,Z 627.416,A -85,B 0,C 180,E1 -13055.595,E2 -13055.595} C_VEL
LIN {X 0,Y 360.659,Z 623.224,A -85,B 0,C 180,E1 -13057.84,E2 -13057.84} C_VEL
LIN {X 0,Y 361.149,Z 617.451,A -85,B 0,C 180,E1 -13060.087,E2 -13060.087} C_VEL
LIN {X 0,Y 361.887,Z 610.924,A -85,B 0,C 180,E1 -13062.05,E2 -13062.05} C_VEL
LIN {X 0,Y 362.751,Z 603.099,A -85,B 0,C 180,E1 -13063.947,E2 -13063.947} C_VEL
LIN {X 0,Y 363.86,Z 594.254,A -85,B 0,C 180,E1 -13065.689,E2 -13065.689} C_VEL
LIN {X 0,Y 365.126,Z 583.877,A -85,B 0,C 180,E1 -13067.358,E2 -13067.358} C_VEL
LIN {X 0,Y 366.446,Z 573.416,A -85,B 0,C 180,E1 -13068.738,E2 -13068.738} C_VEL
LIN {X 0,Y 367.859,Z 562.005,A -85,B 0,C 180,E1 -13069.969,E2 -13069.969} C_VEL
LIN {X 0,Y 369.049,Z 550.031,A -85,B 0,C 180,E1 -13071.019,E2 -13071.019} C_VEL
LIN {X 0,Y 369.964,Z 539.863,A -85,B 0,C 180,E1 -13071.742,E2 -13071.742} C_VEL
LIN {X 0,Y 368.116,Z 527.06,A -85,B 0,C 180,E1 -13072.631,E2 -13072.631} C_VEL
LIN {X 0,Y 365.597,Z 512.743,A -85,B 0,C 180,E1 -13073.421,E2 -13073.421} C_VEL
LIN {X 0,Y 362.461,Z 496.362,A -85,B 0,C 180,E1 -13074.312,E2 -13074.312} C_VEL
LIN {X 0,Y 361.482,Z 491.236,A -85,B 0,C 180,E1 -13074.55,E2 -13074.55} C_VEL
LIN {X 0,Y 361.853,Z 484.452,A -85,B 0,C 180,E1 -13077.784,E2 -13077.784} C_VEL
LIN {X 0,Y 362.28,Z 478.097,A -85,B 0,C 180,E1 -13080.854,E2 -13080.854} C_VEL
LIN {X 0,Y 362.785,Z 471.317,A -85,B 0,C 180,E1 -13084.18,E2 -13084.18} C_VEL
LIN {X 0,Y 363.277,Z 463.244,A -85,B 0,C 180,E1 -13088.249,E2 -13088.249} C_VEL
LIN {X 0,Y 363.791,Z 456.376,A -85,B 0,C 180,E1 -13091.797,E2 -13091.797} C_VEL
LIN {X 0,Y 364.398,Z 449.407,A -85,B 0,C 180,E1 -13095.529,E2 -13095.529} C_VEL
LIN {X 0,Y 364.586,Z 445.689,A -85,B 0,C 180,E1 -13097.57,E2 -13097.57} C_VEL
LIN {X 0,Y 363.97,Z 440.825,A -85,B 0,C 180,E1 -13100.416,E2 -13100.416} C_VEL
LIN {X 0,Y 362.961,Z 435.281,A -85,B 0,C 180,E1 -13103.803,E2 -13103.803} C_VEL
LIN {X 0,Y 362.108,Z 430.186,A -85,B 0,C 180,E1 -13107.082,E2 -13107.082} C_VEL
LIN {X 0,Y 361.879,Z 429.035,A -85,B 0,C 180,E1 -13107.883,E2 -13107.883} C_VEL
LIN {X 0,Y 361.901,Z 429.033,A -85,B 0,C 180,E1 -13110.955,E2 -13110.955} C_VEL
LIN {X 0,Y 361.956,Z 429.01,A -85,B 0,C 180,E1 -13113.475,E2 -13113.475} C_VEL
LIN {X 0,Y 361.892,Z 429.033,A -85,B 0,C 180,E1 -13117.145,E2 -13117.145} C_VEL
LIN {X 0,Y 361.922,Z 429.021,A -85,B 0,C 180,E1 -13120.724,E2 -13120.724} C_VEL
LIN {X 0,Y 361.947,Z 429.015,A -85,B 0,C 180,E1 -13124.226,E2 -13124.226} C_VEL
LIN {X 0,Y 362,Z 429.01,A -85,B 0,C 180,E1 -13126.528,E2 -13126.528} C_VEL
LIN {X 0,Y 362.002,Z 429.009,A -85,B 0,C 180,E1 -13129.937,E2 -13129.937} C_VEL
LIN {X 0,Y 362.153,Z 428.997,A -85,B 0,C 180,E1 -13133.314,E2 -13133.314} C_VEL
LIN {X 0,Y 362.283,Z 428.97,A -85,B 0,C 180,E1 -13137.777,E2 -13137.777} C_VEL
LIN {X 0,Y 362.43,Z 428.967,A -85,B 0,C 180,E1 -13140,E2 -13140} C_VEL
LIN {X 0,Y 362.282,Z 428.972,A -85,B 0,C 180,E1 -13142.224,E2 -13142.224} C_VEL
LIN {X 0,Y 362.174,Z 428.995,A -85,B 0,C 180,E1 -13146.686,E2 -13146.686} C_VEL
LIN {X 0,Y 362.076,Z 428.995,A -85,B 0,C 180,E1 -13148.933,E2 -13148.933} C_VEL
LIN {X 0,Y 361.962,Z 429.02,A -85,B 0,C 180,E1 -13152.332,E2 -13152.332} C_VEL
LIN {X 0,Y 361.964,Z 429.015,A -85,B 0,C 180,E1 -13154.62,E2 -13154.62} C_VEL
LIN {X 0,Y 361.958,Z 429.015,A -85,B 0,C 180,E1 -13158.1,E2 -13158.1} C_VEL
LIN {X 0,Y 361.863,Z 429.034,A -85,B 0,C 180,E1 -13161.655,E2 -13161.655} C_VEL
LIN {X 0,Y 361.929,Z 429.029,A -85,B 0,C 180,E1 -13165.29,E2 -13165.29} C_VEL
LIN {X 0,Y 361.92,Z 429.028,A -85,B 0,C 180,E1 -13167.778,E2 -13167.778} C_VEL
LIN {X 0,Y 361.848,Z 429.038,A -85,B 0,C 180,E1 -13171.285,E2 -13171.285} C_VEL
LIN {X 0,Y 361.856,Z 429.037,A -85,B 0,C 180,E1 -13174.28,E2 -13174.28} C_VEL
LIN {X 0,Y 361.865,Z 429.036,A -85,B 0,C 180,E1 -13177.223,E2 -13177.223} C_VEL
LIN {X 0,Y 361.838,Z 429.043,A -85,B 0,C 180,E1 -13180.756,E2 -13180.756} C_VEL
LIN {X 0,Y 361.864,Z 429.202,A -85,B 0,C 180,E1 -13183.341,E2 -13183.341} C_VEL
LIN {X 0,Y 363.596,Z 437.073,A -85,B 0,C 180,E1 -13186.455,E2 -13186.455} C_VEL
LIN {X 0,Y 364.862,Z 443.842,A -85,B 0,C 180,E1 -13189.087,E2 -13189.087} C_VEL
LIN {X 0,Y 365.296,Z 447.755,A -85,B 0,C 180,E1 -13190.588,E2 -13190.588} C_VEL
LIN {X 0,Y 364.838,Z 455.349,A -85,B 0,C 180,E1 -13193.333,E2 -13193.333} C_VEL
LIN {X 0,Y 364.303,Z 464.631,A -85,B 0,C 180,E1 -13196.663,E2 -13196.663} C_VEL
LIN {X 0,Y 363.805,Z 475.192,A -85,B 0,C 180,E1 -13200.379,E2 -13200.379} C_VEL
LIN {X 0,Y 363.216,Z 486.456,A -85,B 0,C 180,E1 -13204.192,E2 -13204.192} C_VEL
LIN {X 0,Y 363.08,Z 491.488,A -85,B 0,C 180,E1 -13205.78,E2 -13205.78} C_VEL
LIN {X 0,Y 367.071,Z 506.932,A -85,B 0,C 180,E1 -13206.485,E2 -13206.485} C_VEL
LIN {X 0,Y 369.825,Z 520.83,A -85,B 0,C 180,E1 -13207.283,E2 -13207.283} C_VEL
LIN {X 0,Y 370.912,Z 529.711,A -85,B 0,C 180,E1 -13207.871,E2 -13207.871} C_VEL
LIN {X 0,Y 369.835,Z 542.941,A -85,B 0,C 180,E1 -13208.779,E2 -13208.779} C_VEL
LIN {X 0,Y 368.472,Z 555.959,A -85,B 0,C 180,E1 -13209.921,E2 -13209.921} C_VEL
LIN {X 0,Y 367.01,Z 567.263,A -85,B 0,C 180,E1 -13211.147,E2 -13211.147} C_VEL
LIN {X 0,Y 365.594,Z 578.613,A -85,B 0,C 180,E1 -13212.665,E2 -13212.665} C_VEL
LIN {X 0,Y 364.223,Z 588.777,A -85,B 0,C 180,E1 -13214.327,E2 -13214.327} C_VEL
LIN {X 0,Y 363.304,Z 595.837,A -85,B 0,C 180,E1 -13215.721,E2 -13215.721} C_VEL
LIN {X 0,Y 362.446,Z 603.034,A -85,B 0,C 180,E1 -13217.4,E2 -13217.4} C_VEL
LIN {X 0,Y 361.538,Z 609.91,A -85,B 0,C 180,E1 -13219.358,E2 -13219.358} C_VEL
LIN {X 0,Y 360.887,Z 616.075,A -85,B 0,C 180,E1 -13221.602,E2 -13221.602} C_VEL
LIN {X 0,Y 360.611,Z 620.341,A -85,B 0,C 180,E1 -13223.694,E2 -13223.694} C_VEL
LIN {X 0,Y 360.389,Z 623.002,A -85,B 0,C 180,E1 -13225.526,E2 -13225.526} C_VEL
LIN {X 0,Y 360.257,Z 625.036,A -85,B 0,C 180,E1 -13227.764,E2 -13227.764} C_VEL
LIN {X 0,Y 360.274,Z 625.735,A -85,B 0,C 180,E1 -13230,E2 -13230} C_VEL
LIN {X 0,Y 360.256,Z 625.103,A -85,B 0,C 180,E1 -13232.236,E2 -13232.236} C_VEL
LIN {X 0,Y 360.385,Z 623.124,A -85,B 0,C 180,E1 -13234.474,E2 -13234.474} C_VEL
LIN {X 0,Y 360.582,Z 619.763,A -85,B 0,C 180,E1 -13236.716,E2 -13236.716} C_VEL
LIN {X 0,Y 361.018,Z 614.919,A -85,B 0,C 180,E1 -13238.96,E2 -13238.96} C_VEL
LIN {X 0,Y 361.667,Z 608.441,A -85,B 0,C 180,E1 -13241.205,E2 -13241.205} C_VEL
LIN {X 0,Y 362.703,Z 601.217,A -85,B 0,C 180,E1 -13243.16,E2 -13243.16} C_VEL
LIN {X 0,Y 363.671,Z 593.215,A -85,B 0,C 180,E1 -13244.926,E2 -13244.926} C_VEL
LIN {X 0,Y 365.063,Z 582.806,A -85,B 0,C 180,E1 -13246.784,E2 -13246.784} C_VEL
LIN {X 0,Y 366.415,Z 572.379,A -85,B 0,C 180,E1 -13248.305,E2 -13248.305} C_VEL
LIN {X 0,Y 367.888,Z 560.867,A -85,B 0,C 180,E1 -13249.676,E2 -13249.676} C_VEL
LIN {X 0,Y 369.345,Z 548.099,A -85,B 0,C 180,E1 -13250.903,E2 -13250.903} C_VEL
LIN {X 0,Y 370.604,Z 534.518,A -85,B 0,C 180,E1 -13251.927,E2 -13251.927} C_VEL
LIN {X 0,Y 370.887,Z 527.922,A -85,B 0,C 180,E1 -13252.345,E2 -13252.345} C_VEL
LIN {X 0,Y 368.785,Z 514.853,A -85,B 0,C 180,E1 -13253.181,E2 -13253.181} C_VEL
LIN {X 0,Y 365.537,Z 500.572,A -85,B 0,C 180,E1 -13253.928,E2 -13253.928} C_VEL
LIN {X 0,Y 364.72,Z 497.606,A -85,B 0,C 180,E1 -13254.067,E2 -13254.067} C_VEL
LIN {X 0,Y 363.623,Z 494.401,A -85,B 0,C 180,E1 -13254.317,E2 -13254.317} C_VEL
LIN {X 0,Y 361.941,Z 491.236,A -85,B 0,C 180,E1 -13254.808,E2 -13254.808} C_VEL
LIN {X 0,Y 359.59,Z 487.988,A -85,B 0,C 180,E1 -13255.68,E2 -13255.68} C_VEL
LIN {X 0,Y 357.377,Z 484.892,A -85,B 0,C 180,E1 -13256.882,E2 -13256.882} C_VEL
LIN {X 0,Y 356.598,Z 482.381,A -85,B 0,C 180,E1 -13257.812,E2 -13257.812} C_VEL
LIN {X 0,Y 356.574,Z 481.492,A -85,B 0,C 180,E1 -13258.122,E2 -13258.122} C_VEL
LIN {X 0,Y 357.075,Z 471.952,A -85,B 0,C 180,E1 -13261.438,E2 -13261.438} C_VEL
LIN {X 0,Y 357.623,Z 462.747,A -85,B 0,C 180,E1 -13264.744,E2 -13264.744} C_VEL
LIN {X 0,Y 358.411,Z 451.483,A -85,B 0,C 180,E1 -13268.865,E2 -13268.865} C_VEL
LIN {X 0,Y 358.278,Z 447.557,A -85,B 0,C 180,E1 -13270.341,E2 -13270.341} C_VEL
LIN {X 0,Y 356.832,Z 439.387,A -85,B 0,C 180,E1 -13273.578,E2 -13273.578} C_VEL
LIN {X 0,Y 355.146,Z 431.567,A -85,B 0,C 180,E1 -13276.722,E2 -13276.722} C_VEL
LIN {X 0,Y 354.791,Z 429.925,A -85,B 0,C 180,E1 -13277.446,E2 -13277.446} C_VEL
LIN {X 0,Y 354.816,Z 429.914,A -85,B 0,C 180,E1 -13280.666,E2 -13280.666} C_VEL
LIN {X 0,Y 354.824,Z 429.914,A -85,B 0,C 180,E1 -13284.301,E2 -13284.301} C_VEL
LIN {X 0,Y 354.789,Z 429.918,A -85,B 0,C 180,E1 -13287.667,E2 -13287.667} C_VEL
LIN {X 0,Y 354.87,Z 429.901,A -85,B 0,C 180,E1 -13290.621,E2 -13290.621} C_VEL
LIN {X 0,Y 354.915,Z 429.9,A -85,B 0,C 180,E1 -13294.306,E2 -13294.306} C_VEL
LIN {X 0,Y 359.807,Z 445.009,A -85,B 0,C 180,E1 -13295.583,E2 -13295.583} C_VEL
LIN {X 0,Y 363.535,Z 457.106,A -85,B 0,C 180,E1 -13296.767,E2 -13296.767} C_VEL
LIN {X 0,Y 362.501,Z 469.798,A -85,B 0,C 180,E1 -13297.936,E2 -13297.936} C_VEL
LIN {X 0,Y 361.136,Z 482.513,A -85,B 0,C 180,E1 -13299.333,E2 -13299.333} C_VEL
LIN {X 0,Y 359.776,Z 494.428,A -85,B 0,C 180,E1 -13300.901,E2 -13300.901} C_VEL
LIN {X 0,Y 358.526,Z 505.285,A -85,B 0,C 180,E1 -13302.606,E2 -13302.606} C_VEL
LIN {X 0,Y 357.291,Z 515.141,A -85,B 0,C 180,E1 -13304.446,E2 -13304.446} C_VEL
LIN {X 0,Y 356.483,Z 523.503,A -85,B 0,C 180,E1 -13306.315,E2 -13306.315} C_VEL
LIN {X 0,Y 355.705,Z 530.048,A -85,B 0,C 180,E1 -13308.026,E2 -13308.026} C_VEL
LIN {X 0,Y 355.018,Z 537.169,A -85,B 0,C 180,E1 -13310.313,E2 -13310.313} C_VEL
LIN {X 0,Y 354.577,Z 542.169,A -85,B 0,C 180,E1 -13312.324,E2 -13312.324} C_VEL
LIN {X 0,Y 354.34,Z 546.004,A -85,B 0,C 180,E1 -13314.309,E2 -13314.309} C_VEL
LIN {X 0,Y 354.19,Z 549.224,A -85,B 0,C 180,E1 -13316.587,E2 -13316.587} C_VEL
LIN {X 0,Y 353.841,Z 551.237,A -85,B 0,C 180,E1 -13318.862,E2 -13318.862} C_VEL
LIN {X 0,Y 353.881,Z 552.026,A -85,B 0,C 180,E1 -13321.138,E2 -13321.138} C_VEL
LIN {X 0,Y 354.226,Z 551.605,A -85,B 0,C 180,E1 -13323.412,E2 -13323.412} C_VEL
LIN {X 0,Y 354.825,Z 549.972,A -85,B 0,C 180,E1 -13325.684,E2 -13325.684} C_VEL
LIN {X 0,Y 355.345,Z 547.134,A -85,B 0,C 180,E1 -13327.958,E2 -13327.958} C_VEL
LIN {X 0,Y 356.184,Z 542.994,A -85,B 0,C 180,E1 -13330.229,E2 -13330.229} C_VEL
LIN {X 0,Y 357.058,Z 537.469,A -85,B 0,C 180,E1 -13332.504,E2 -13332.504} C_VEL
LIN {X 0,Y 358.488,Z 530.294,A -85,B 0,C 180,E1 -13334.765,E2 -13334.765} C_VEL
LIN {X 0,Y 359.921,Z 523.113,A -85,B 0,C 180,E1 -13336.619,E2 -13336.619} C_VEL
LIN {X 0,Y 361.469,Z 514.714,A -85,B 0,C 180,E1 -13338.418,E2 -13338.418} C_VEL
LIN {X 0,Y 363.384,Z 503.691,A -85,B 0,C 180,E1 -13340.373,E2 -13340.373} C_VEL
LIN {X 0,Y 365.219,Z 492.798,A -85,B 0,C 180,E1 -13341.964,E2 -13341.964} C_VEL
LIN {X 0,Y 367.344,Z 479.64,A -85,B 0,C 180,E1 -13343.543,E2 -13343.543} C_VEL
LIN {X 0,Y 368.981,Z 467.342,A -85,B 0,C 180,E1 -13344.774,E2 -13344.774} C_VEL
LIN {X 0,Y 369.474,Z 463.908,A -85,B 0,C 180,E1 -13345.074,E2 -13345.074} C_VEL
LIN {X 0,Y 368.483,Z 459.547,A -85,B 0,C 180,E1 -13345.622,E2 -13345.622} C_VEL
LIN {X 0,Y 365.315,Z 450.648,A -85,B 0,C 180,E1 -13346.831,E2 -13346.831} C_VEL
LIN {X 0,Y 360.585,Z 440.642,A -85,B 0,C 180,E1 -13348.316,E2 -13348.316} C_VEL
LIN {X 0,Y 357.014,Z 434.153,A -85,B 0,C 180,E1 -13349.352,E2 -13349.352} C_VEL
LIN {X 0,Y 355.306,Z 431.665,A -85,B 0,C 180,E1 -13349.816,E2 -13349.816} C_VEL
LIN {X 0,Y 354.838,Z 429.913,A -85,B 0,C 180,E1 -13350.041,E2 -13350.041} C_VEL
LIN {X 0,Y 354.807,Z 429.916,A -85,B 0,C 180,E1 -13353.702,E2 -13353.702} C_VEL
LIN {X 0,Y 354.829,Z 429.959,A -85,B 0,C 180,E1 -13357.188,E2 -13357.188} C_VEL
LIN {X 0,Y 355.568,Z 434.025,A -85,B 0,C 180,E1 -13360.713,E2 -13360.713} C_VEL
LIN {X 0,Y 356.123,Z 438.209,A -85,B 0,C 180,E1 -13363.687,E2 -13363.687} C_VEL
LIN {X 0,Y 355.858,Z 440.888,A -85,B 0,C 180,E1 -13365.315,E2 -13365.315} C_VEL
LIN {X 0,Y 355.129,Z 449.318,A -85,B 0,C 180,E1 -13369.937,E2 -13369.937} C_VEL
LIN {X 0,Y 354.905,Z 456.57,A -85,B 0,C 180,E1 -13373.553,E2 -13373.553} C_VEL
LIN {X 0,Y 354.643,Z 463.902,A -85,B 0,C 180,E1 -13376.989,E2 -13376.989} C_VEL
LIN {X 0,Y 354.448,Z 472.246,A -85,B 0,C 180,E1 -13380.743,E2 -13380.743} C_VEL
LIN {X 0,Y 354.367,Z 474.957,A -85,B 0,C 180,E1 -13381.939,E2 -13381.939} C_VEL
LIN {X 0,Y 355.052,Z 478.583,A -85,B 0,C 180,E1 -13382.237,E2 -13382.237} C_VEL
LIN {X 0,Y 356.072,Z 481.281,A -85,B 0,C 180,E1 -13382.532,E2 -13382.532} C_VEL
LIN {X 0,Y 357.24,Z 485.552,A -85,B 0,C 180,E1 -13382.922,E2 -13382.922} C_VEL
LIN {X 0,Y 360.267,Z 499.629,A -85,B 0,C 180,E1 -13384.175,E2 -13384.175} C_VEL
LIN {X 0,Y 361.988,Z 513.612,A -85,B 0,C 180,E1 -13385.379,E2 -13385.379} C_VEL
LIN {X 0,Y 362.377,Z 530.123,A -85,B 0,C 180,E1 -13386.848,E2 -13386.848} C_VEL
LIN {X 0,Y 363.107,Z 539.945,A -85,B 0,C 180,E1 -13387.826,E2 -13387.826} C_VEL
LIN {X 0,Y 363.044,Z 543.949,A -85,B 0,C 180,E1 -13388.121,E2 -13388.121} C_VEL
LIN {X 0,Y 361.795,Z 556.45,A -85,B 0,C 180,E1 -13389.119,E2 -13389.119} C_VEL
LIN {X 0,Y 360.427,Z 568.651,A -85,B 0,C 180,E1 -13390.345,E2 -13390.345} C_VEL
LIN {X 0,Y 358.916,Z 579.954,A -85,B 0,C 180,E1 -13391.742,E2 -13391.742} C_VEL
LIN {X 0,Y 357.44,Z 590.986,A -85,B 0,C 180,E1 -13393.435,E2 -13393.435} C_VEL
LIN {X 0,Y 356.237,Z 600.21,A -85,B 0,C 180,E1 -13395.171,E2 -13395.171} C_VEL
LIN {X 0,Y 355.202,Z 608.719,A -85,B 0,C 180,E1 -13397.139,E2 -13397.139} C_VEL
LIN {X 0,Y 354.297,Z 615.687,A -85,B 0,C 180,E1 -13399.138,E2 -13399.138} C_VEL
LIN {X 0,Y 353.848,Z 620.501,A -85,B 0,C 180,E1 -13400.857,E2 -13400.857} C_VEL
LIN {X 0,Y 353.501,Z 625.458,A -85,B 0,C 180,E1 -13403.149,E2 -13403.149} C_VEL
LIN {X 0,Y 353.329,Z 628.903,A -85,B 0,C 180,E1 -13405.437,E2 -13405.437} C_VEL
LIN {X 0,Y 353.231,Z 630.943,A -85,B 0,C 180,E1 -13407.719,E2 -13407.719} C_VEL
LIN {X 0,Y 353.248,Z 631.621,A -85,B 0,C 180,E1 -13410,E2 -13410} C_VEL
LIN {X 0,Y 353.231,Z 630.941,A -85,B 0,C 180,E1 -13412.281,E2 -13412.281} C_VEL
LIN {X 0,Y 353.313,Z 628.901,A -85,B 0,C 180,E1 -13414.564,E2 -13414.564} C_VEL
LIN {X 0,Y 353.432,Z 625.45,A -85,B 0,C 180,E1 -13416.852,E2 -13416.852} C_VEL
LIN {X 0,Y 353.835,Z 620.486,A -85,B 0,C 180,E1 -13419.143,E2 -13419.143} C_VEL
LIN {X 0,Y 354.291,Z 615.668,A -85,B 0,C 180,E1 -13420.862,E2 -13420.862} C_VEL
LIN {X 0,Y 355.172,Z 608.697,A -85,B 0,C 180,E1 -13422.862,E2 -13422.862} C_VEL
LIN {X 0,Y 356.167,Z 600.033,A -85,B 0,C 180,E1 -13424.864,E2 -13424.864} C_VEL
LIN {X 0,Y 357.415,Z 590.951,A -85,B 0,C 180,E1 -13426.566,E2 -13426.566} C_VEL
LIN {X 0,Y 358.871,Z 579.907,A -85,B 0,C 180,E1 -13428.261,E2 -13428.261} C_VEL
LIN {X 0,Y 360.407,Z 568.592,A -85,B 0,C 180,E1 -13429.656,E2 -13429.656} C_VEL
LIN {X 0,Y 361.782,Z 556.557,A -85,B 0,C 180,E1 -13430.865,E2 -13430.865} C_VEL
LIN {X 0,Y 362.99,Z 543.849,A -85,B 0,C 180,E1 -13431.883,E2 -13431.883} C_VEL
LIN {X 0,Y 363.109,Z 539.826,A -85,B 0,C 180,E1 -13432.174,E2 -13432.174} C_VEL
LIN {X 0,Y 361.438,Z 527.74,A -85,B 0,C 180,E1 -13433.037,E2 -13433.037} C_VEL
LIN {X 0,Y 358.894,Z 513.44,A -85,B 0,C 180,E1 -13433.858,E2 -13433.858} C_VEL
LIN {X 0,Y 354.456,Z 490.51,A -85,B 0,C 180,E1 -13435.029,E2 -13435.029} C_VEL
LIN {X 0,Y 354.957,Z 482.571,A -85,B 0,C 180,E1 -13438.903,E2 -13438.903} C_VEL
LIN {X 0,Y 355.423,Z 475.784,A -85,B 0,C 180,E1 -13442.269,E2 -13442.269} C_VEL
LIN {X 0,Y 355.779,Z 470.458,A -85,B 0,C 180,E1 -13444.95,E2 -13444.95} C_VEL
LIN {X 0,Y 356.251,Z 463.625,A -85,B 0,C 180,E1 -13448.46,E2 -13448.46} C_VEL
LIN {X 0,Y 356.774,Z 456.837,A -85,B 0,C 180,E1 -13452.048,E2 -13452.048} C_VEL
LIN {X 0,Y 357.285,Z 451.242,A -85,B 0,C 180,E1 -13455.084,E2 -13455.084} C_VEL
LIN {X 0,Y 357.507,Z 445.947,A -85,B 0,C 180,E1 -13458.058,E2 -13458.058} C_VEL
LIN {X 0,Y 356.829,Z 441.136,A -85,B 0,C 180,E1 -13460.93,E2 -13460.93} C_VEL
LIN {X 0,Y 355.9,Z 436.146,A -85,B 0,C 180,E1 -13464.06,E2 -13464.06} C_VEL
LIN {X 0,Y 354.971,Z 430.6,A -85,B 0,C 180,E1 -13467.685,E2 -13467.685} C_VEL
LIN {X 0,Y 354.826,Z 429.914,A -85,B 0,C 180,E1 -13468.294,E2 -13468.294} C_VEL
LIN {X 0,Y 354.852,Z 429.909,A -85,B 0,C 180,E1 -13471.619,E2 -13471.619} C_VEL
LIN {X 0,Y 354.901,Z 429.888,A -85,B 0,C 180,E1 -13474.173,E2 -13474.173} C_VEL
LIN {X 0,Y 354.836,Z 429.906,A -85,B 0,C 180,E1 -13477.894,E2 -13477.894} C_VEL
LIN {X 0,Y 354.924,Z 429.9,A -85,B 0,C 180,E1 -13481.891,E2 -13481.891} C_VEL
LIN {X 0,Y 354.944,Z 429.885,A -85,B 0,C 180,E1 -13485.981,E2 -13485.981} C_VEL
LIN {X 0,Y 354.958,Z 429.887,A -85,B 0,C 180,E1 -13489.735,E2 -13489.735} C_VEL
LIN {X 0,Y 355.116,Z 429.874,A -85,B 0,C 180,E1 -13493.18,E2 -13493.18} C_VEL
LIN {X 0,Y 355.246,Z 429.845,A -85,B 0,C 180,E1 -13497.732,E2 -13497.732} C_VEL
LIN {X 0,Y 355.4,Z 429.843,A -85,B 0,C 180,E1 -13500,E2 -13500} C_VEL
LIN {X 0,Y 355.245,Z 429.847,A -85,B 0,C 180,E1 -13502.268,E2 -13502.268} C_VEL
LIN {X 0,Y 355.14,Z 429.871,A -85,B 0,C 180,E1 -13506.819,E2 -13506.819} C_VEL
LIN {X 0,Y 355.017,Z 429.875,A -85,B 0,C 180,E1 -13509.112,E2 -13509.112} C_VEL
LIN {X 0,Y 354.923,Z 429.895,A -85,B 0,C 180,E1 -13512.581,E2 -13512.581} C_VEL
LIN {X 0,Y 354.892,Z 429.905,A -85,B 0,C 180,E1 -13516.096,E2 -13516.096} C_VEL
LIN {X 0,Y 354.903,Z 429.891,A -85,B 0,C 180,E1 -13518.472,E2 -13518.472} C_VEL
LIN {X 0,Y 354.818,Z 429.909,A -85,B 0,C 180,E1 -13522.107,E2 -13522.107} C_VEL
LIN {X 0,Y 354.9,Z 429.899,A -85,B 0,C 180,E1 -13525.827,E2 -13525.827} C_VEL
LIN {X 0,Y 354.855,Z 429.904,A -85,B 0,C 180,E1 -13529.679,E2 -13529.679} C_VEL
LIN {X 0,Y 354.807,Z 429.913,A -85,B 0,C 180,E1 -13533.702,E2 -13533.702} C_VEL
LIN {X 0,Y 354.8,Z 429.916,A -85,B 0,C 180,E1 -13536.459,E2 -13536.459} C_VEL
LIN {X 0,Y 354.825,Z 429.912,A -85,B 0,C 180,E1 -13539.424,E2 -13539.424} C_VEL
LIN {X 0,Y 354.818,Z 430.016,A -85,B 0,C 180,E1 -13542.774,E2 -13542.774} C_VEL
LIN {X 0,Y 356.799,Z 439.065,A -85,B 0,C 180,E1 -13546.417,E2 -13546.417} C_VEL
LIN {X 0,Y 357.974,Z 445.519,A -85,B 0,C 180,E1 -13548.986,E2 -13548.986} C_VEL
LIN {X 0,Y 358.406,Z 451.163,A -85,B 0,C 180,E1 -13551.135,E2 -13551.135} C_VEL
LIN {X 0,Y 357.625,Z 462.458,A -85,B 0,C 180,E1 -13555.256,E2 -13555.256} C_VEL
LIN {X 0,Y 357.027,Z 473.519,A -85,B 0,C 180,E1 -13559.216,E2 -13559.216} C_VEL
LIN {X 0,Y 356.468,Z 483.051,A -85,B 0,C 180,E1 -13562.524,E2 -13562.524} C_VEL
LIN {X 0,Y 356.138,Z 491.369,A -85,B 0,C 180,E1 -13565.275,E2 -13565.275} C_VEL
LIN {X 0,Y 360.209,Z 506.779,A -85,B 0,C 180,E1 -13566.003,E2 -13566.003} C_VEL
LIN {X 0,Y 363.01,Z 520.917,A -85,B 0,C 180,E1 -13566.836,E2 -13566.836} C_VEL
LIN {X 0,Y 364.322,Z 529.85,A -85,B 0,C 180,E1 -13567.456,E2 -13567.456} C_VEL
LIN {X 0,Y 363.298,Z 541.927,A -85,B 0,C 180,E1 -13568.286,E2 -13568.286} C_VEL
LIN {X 0,Y 361.98,Z 554.617,A -85,B 0,C 180,E1 -13569.396,E2 -13569.396} C_VEL
LIN {X 0,Y 360.462,Z 566.166,A -85,B 0,C 180,E1 -13570.643,E2 -13570.643} C_VEL
LIN {X 0,Y 359.034,Z 576.753,A -85,B 0,C 180,E1 -13572.043,E2 -13572.043} C_VEL
LIN {X 0,Y 357.591,Z 587.238,A -85,B 0,C 180,E1 -13573.736,E2 -13573.736} C_VEL
LIN {X 0,Y 356.36,Z 595.895,A -85,B 0,C 180,E1 -13575.437,E2 -13575.437} C_VEL
LIN {X 0,Y 355.5,Z 603.091,A -85,B 0,C 180,E1 -13577.15,E2 -13577.15} C_VEL
LIN {X 0,Y 354.531,Z 609.969,A -85,B 0,C 180,E1 -13579.145,E2 -13579.145} C_VEL
LIN {X 0,Y 353.837,Z 616.134,A -85,B 0,C 180,E1 -13581.433,E2 -13581.433} C_VEL
LIN {X 0,Y 353.513,Z 620.665,A -85,B 0,C 180,E1 -13583.734,E2 -13583.734} C_VEL
LIN {X 0,Y 353.306,Z 623.061,A -85,B 0,C 180,E1 -13585.436,E2 -13585.436} C_VEL
LIN {X 0,Y 353.165,Z 625.095,A -85,B 0,C 180,E1 -13587.719,E2 -13587.719} C_VEL
LIN {X 0,Y 353.174,Z 625.794,A -85,B 0,C 180,E1 -13590,E2 -13590} C_VEL
LIN {X 0,Y 353.165,Z 625.161,A -85,B 0,C 180,E1 -13592.281,E2 -13592.281} C_VEL
LIN {X 0,Y 353.301,Z 623.182,A -85,B 0,C 180,E1 -13594.564,E2 -13594.564} C_VEL
LIN {X 0,Y 353.518,Z 619.82,A -85,B 0,C 180,E1 -13596.851,E2 -13596.851} C_VEL
LIN {X 0,Y 353.964,Z 614.975,A -85,B 0,C 180,E1 -13599.14,E2 -13599.14} C_VEL
LIN {X 0,Y 354.664,Z 608.496,A -85,B 0,C 180,E1 -13601.429,E2 -13601.429} C_VEL
LIN {X 0,Y 355.772,Z 601.27,A -85,B 0,C 180,E1 -13603.421,E2 -13603.421} C_VEL
LIN {X 0,Y 356.925,Z 592.274,A -85,B 0,C 180,E1 -13605.415,E2 -13605.415} C_VEL
LIN {X 0,Y 358.237,Z 582.854,A -85,B 0,C 180,E1 -13607.114,E2 -13607.114} C_VEL
LIN {X 0,Y 359.638,Z 572.425,A -85,B 0,C 180,E1 -13608.663,E2 -13608.663} C_VEL
LIN {X 0,Y 361.183,Z 560.907,A -85,B 0,C 180,E1 -13610.057,E2 -13610.057} C_VEL
LIN {X 0,Y 362.721,Z 548.133,A -85,B 0,C 180,E1 -13611.303,E2 -13611.303} C_VEL
LIN {X 0,Y 364.01,Z 534.61,A -85,B 0,C 180,E1 -13612.34,E2 -13612.34} C_VEL
LIN {X 0,Y 364.258,Z 529.159,A -85,B 0,C 180,E1 -13612.698,E2 -13612.698} C_VEL
LIN {X 0,Y 362.145,Z 515.725,A -85,B 0,C 180,E1 -13613.593,E2 -13613.593} C_VEL
LIN {X 0,Y 358.941,Z 501.764,A -85,B 0,C 180,E1 -13614.361,E2 -13614.361} C_VEL
LIN {X 0,Y 356.114,Z 491.21,A -85,B 0,C 180,E1 -13614.863,E2 -13614.863} C_VEL
LIN {X 0,Y 356.574,Z 481.492,A -85,B 0,C 180,E1 -13618.122,E2 -13618.122} C_VEL
LIN {X 0,Y 356.038,Z 479.133,A -85,B 0,C 180,E1 -13618.988,E2 -13618.988} C_VEL
LIN {X 0,Y 353.422,Z 475.675,A -85,B 0,C 180,E1 -13620.429,E2 -13620.429} C_VEL
LIN {X 0,Y 351.223,Z 472.964,A -85,B 0,C 180,E1 -13621.598,E2 -13621.598} C_VEL
LIN {X 0,Y 350.362,Z 470.74,A -85,B 0,C 180,E1 -13622.489,E2 -13622.489} C_VEL
LIN {X 0,Y 350.338,Z 469.935,A -85,B 0,C 180,E1 -13622.785,E2 -13622.785} C_VEL
LIN {X 0,Y 350.916,Z 460.722,A -85,B 0,C 180,E1 -13626.155,E2 -13626.155} C_VEL
LIN {X 0,Y 351.573,Z 452.603,A -85,B 0,C 180,E1 -13629.177,E2 -13629.177} C_VEL
LIN {X 0,Y 351.073,Z 446.999,A -85,B 0,C 180,E1 -13631.347,E2 -13631.347} C_VEL
LIN {X 0,Y 349.472,Z 438.645,A -85,B 0,C 180,E1 -13634.738,E2 -13634.738} C_VEL
LIN {X 0,Y 347.749,Z 430.798,A -85,B 0,C 180,E1 -13637.975,E2 -13637.975} C_VEL
LIN {X 0,Y 347.776,Z 430.794,A -85,B 0,C 180,E1 -13642.011,E2 -13642.011} C_VEL
LIN {X 0,Y 347.746,Z 430.787,A -85,B 0,C 180,E1 -13645.536,E2 -13645.536} C_VEL
LIN {X 0,Y 347.766,Z 430.779,A -85,B 0,C 180,E1 -13649.654,E2 -13649.654} C_VEL
LIN {X 0,Y 347.854,Z 430.782,A -85,B 0,C 180,E1 -13652.744,E2 -13652.744} C_VEL
LIN {X 0,Y 347.861,Z 430.78,A -85,B 0,C 180,E1 -13653.919,E2 -13653.919} C_VEL
LIN {X 0,Y 352.91,Z 446.29,A -85,B 0,C 180,E1 -13655.279,E2 -13655.279} C_VEL
LIN {X 0,Y 356.786,Z 459.409,A -85,B 0,C 180,E1 -13656.6,E2 -13656.6} C_VEL
LIN {X 0,Y 355.342,Z 473.281,A -85,B 0,C 180,E1 -13657.927,E2 -13657.927} C_VEL
LIN {X 0,Y 353.871,Z 486.784,A -85,B 0,C 180,E1 -13659.51,E2 -13659.51} C_VEL
LIN {X 0,Y 352.558,Z 498.087,A -85,B 0,C 180,E1 -13661.099,E2 -13661.099} C_VEL
LIN {X 0,Y 351.306,Z 508.508,A -85,B 0,C 180,E1 -13662.838,E2 -13662.838} C_VEL
LIN {X 0,Y 350.006,Z 518.685,A -85,B 0,C 180,E1 -13664.868,E2 -13664.868} C_VEL
LIN {X 0,Y 349.243,Z 526.015,A -85,B 0,C 180,E1 -13666.619,E2 -13666.619} C_VEL
LIN {X 0,Y 348.355,Z 534.157,A -85,B 0,C 180,E1 -13668.95,E2 -13668.95} C_VEL
LIN {X 0,Y 347.709,Z 540.612,A -85,B 0,C 180,E1 -13671.281,E2 -13671.281} C_VEL
LIN {X 0,Y 347.279,Z 545.591,A -85,B 0,C 180,E1 -13673.609,E2 -13673.609} C_VEL
LIN {X 0,Y 347.228,Z 548.384,A -85,B 0,C 180,E1 -13675.356,E2 -13675.356} C_VEL
LIN {X 0,Y 347.156,Z 549.879,A -85,B 0,C 180,E1 -13676.518,E2 -13676.518} C_VEL
LIN {X 0,Y 346.795,Z 551.981,A -85,B 0,C 180,E1 -13678.839,E2 -13678.839} C_VEL
LIN {X 0,Y 346.832,Z 552.861,A -85,B 0,C 180,E1 -13681.161,E2 -13681.161} C_VEL
LIN {X 0,Y 347.199,Z 552.522,A -85,B 0,C 180,E1 -13683.481,E2 -13683.481} C_VEL
LIN {X 0,Y 347.827,Z 550.966,A -85,B 0,C 180,E1 -13685.798,E2 -13685.798} C_VEL
LIN {X 0,Y 348.393,Z 548.221,A -85,B 0,C 180,E1 -13688.118,E2 -13688.118} C_VEL
LIN {X 0,Y 349.287,Z 544.157,A -85,B 0,C 180,E1 -13690.433,E2 -13690.433} C_VEL
LIN {X 0,Y 350.239,Z 538.738,A -85,B 0,C 180,E1 -13692.752,E2 -13692.752} C_VEL
LIN {X 0,Y 351.775,Z 531.725,A -85,B 0,C 180,E1 -13695.054,E2 -13695.054} C_VEL
LIN {X 0,Y 352.916,Z 526.086,A -85,B 0,C 180,E1 -13696.573,E2 -13696.573} C_VEL
LIN {X 0,Y 354.647,Z 517.735,A -85,B 0,C 180,E1 -13698.486,E2 -13698.486} C_VEL
LIN {X 0,Y 356.334,Z 508.857,A -85,B 0,C 180,E1 -13700.191,E2 -13700.191} C_VEL
LIN {X 0,Y 358.644,Z 496.426,A -85,B 0,C 180,E1 -13702.162,E2 -13702.162} C_VEL
LIN {X 0,Y 360.875,Z 484.047,A -85,B 0,C 180,E1 -13703.749,E2 -13703.749} C_VEL
LIN {X 0,Y 362.923,Z 470.185,A -85,B 0,C 180,E1 -13705.216,E2 -13705.216} C_VEL
LIN {X 0,Y 363.534,Z 466.076,A -85,B 0,C 180,E1 -13705.598,E2 -13705.598} C_VEL
LIN {X 0,Y 360.979,Z 457.294,A -85,B 0,C 180,E1 -13706.826,E2 -13706.826} C_VEL
LIN {X 0,Y 356.824,Z 447.343,A -85,B 0,C 180,E1 -13708.356,E2 -13708.356} C_VEL
LIN {X 0,Y 352.508,Z 439.244,A -85,B 0,C 180,E1 -13709.744,E2 -13709.744} C_VEL
LIN {X 0,Y 350.665,Z 436.051,A -85,B 0,C 180,E1 -13710.321,E2 -13710.321} C_VEL
LIN {X 0,Y 350.417,Z 435.447,A -85,B 0,C 180,E1 -13710.411,E2 -13710.411} C_VEL
LIN {X 0,Y 348.455,Z 433.042,A -85,B 0,C 180,E1 -13710.983,E2 -13710.983} C_VEL
LIN {X 0,Y 347.748,Z 430.796,A -85,B 0,C 180,E1 -13711.305,E2 -13711.305} C_VEL
LIN {X 0,Y 347.745,Z 430.794,A -85,B 0,C 180,E1 -13714.464,E2 -13714.464} C_VEL
LIN {X 0,Y 347.795,Z 430.891,A -85,B 0,C 180,E1 -13716.466,E2 -13716.466} C_VEL
LIN {X 0,Y 348.228,Z 433.222,A -85,B 0,C 180,E1 -13718.73,E2 -13718.73} C_VEL
LIN {X 0,Y 348.885,Z 436.991,A -85,B 0,C 180,E1 -13721.812,E2 -13721.812} C_VEL
LIN {X 0,Y 349.177,Z 439.462,A -85,B 0,C 180,E1 -13723.566,E2 -13723.566} C_VEL
LIN {X 0,Y 348.695,Z 443.265,A -85,B 0,C 180,E1 -13725.914,E2 -13725.914} C_VEL
LIN {X 0,Y 348.1,Z 450.764,A -85,B 0,C 180,E1 -13730.104,E2 -13730.104} C_VEL
LIN {X 0,Y 347.819,Z 458.671,A -85,B 0,C 180,E1 -13734.128,E2 -13734.128} C_VEL
LIN {X 0,Y 347.516,Z 467.11,A -85,B 0,C 180,E1 -13738.145,E2 -13738.145} C_VEL
LIN {X 0,Y 347.366,Z 472.734,A -85,B 0,C 180,E1 -13740.729,E2 -13740.729} C_VEL
LIN {X 0,Y 348.171,Z 476.704,A -85,B 0,C 180,E1 -13741.105,E2 -13741.105} C_VEL
LIN {X 0,Y 349.272,Z 479.656,A -85,B 0,C 180,E1 -13741.46,E2 -13741.46} C_VEL
LIN {X 0,Y 351.085,Z 486.52,A -85,B 0,C 180,E1 -13742.161,E2 -13742.161} C_VEL
LIN {X 0,Y 353.489,Z 496.844,A -85,B 0,C 180,E1 -13743.185,E2 -13743.185} C_VEL
LIN {X 0,Y 355.292,Z 509.39,A -85,B 0,C 180,E1 -13744.356,E2 -13744.356} C_VEL
LIN {X 0,Y 355.924,Z 520.305,A -85,B 0,C 180,E1 -13745.352,E2 -13745.352} C_VEL
LIN {X 0,Y 356.013,Z 534.485,A -85,B 0,C 180,E1 -13746.745,E2 -13746.745} C_VEL
LIN {X 0,Y 356.526,Z 541.946,A -85,B 0,C 180,E1 -13747.547,E2 -13747.547} C_VEL
LIN {X 0,Y 355.441,Z 553.81,A -85,B 0,C 180,E1 -13748.476,E2 -13748.476} C_VEL
LIN {X 0,Y 354.015,Z 566.034,A -85,B 0,C 180,E1 -13749.671,E2 -13749.671} C_VEL
LIN {X 0,Y 352.398,Z 577.778,A -85,B 0,C 180,E1 -13751.09,E2 -13751.09} C_VEL
LIN {X 0,Y 351.114,Z 587.484,A -85,B 0,C 180,E1 -13752.528,E2 -13752.528} C_VEL
LIN {X 0,Y 349.712,Z 597.169,A -85,B 0,C 180,E1 -13754.258,E2 -13754.258} C_VEL
LIN {X 0,Y 348.537,Z 606.411,A -85,B 0,C 180,E1 -13756.295,E2 -13756.295} C_VEL
LIN {X 0,Y 347.482,Z 613.823,A -85,B 0,C 180,E1 -13758.331,E2 -13758.331} C_VEL
LIN {X 0,Y 346.955,Z 618.966,A -85,B 0,C 180,E1 -13760.086,E2 -13760.086} C_VEL
LIN {X 0,Y 346.545,Z 623.12,A -85,B 0,C 180,E1 -13761.839,E2 -13761.839} C_VEL
LIN {X 0,Y 346.288,Z 627.304,A -85,B 0,C 180,E1 -13764.176,E2 -13764.176} C_VEL
LIN {X 0,Y 346.181,Z 630.036,A -85,B 0,C 180,E1 -13766.508,E2 -13766.508} C_VEL
LIN {X 0,Y 346.142,Z 631.393,A -85,B 0,C 180,E1 -13768.837,E2 -13768.837} C_VEL
LIN {X 0,Y 346.142,Z 631.392,A -85,B 0,C 180,E1 -13771.163,E2 -13771.163} C_VEL
LIN {X 0,Y 346.178,Z 630.034,A -85,B 0,C 180,E1 -13773.492,E2 -13773.492} C_VEL
LIN {X 0,Y 346.248,Z 627.298,A -85,B 0,C 180,E1 -13775.825,E2 -13775.825} C_VEL
LIN {X 0,Y 346.541,Z 623.107,A -85,B 0,C 180,E1 -13778.161,E2 -13778.161} C_VEL
LIN {X 0,Y 347.1,Z 617.334,A -85,B 0,C 180,E1 -13780.5,E2 -13780.5} C_VEL
LIN {X 0,Y 347.935,Z 610.809,A -85,B 0,C 180,E1 -13782.541,E2 -13782.541} C_VEL
LIN {X 0,Y 348.794,Z 603.768,A -85,B 0,C 180,E1 -13784.328,E2 -13784.328} C_VEL
LIN {X 0,Y 349.906,Z 595.65,A -85,B 0,C 180,E1 -13786.032,E2 -13786.032} C_VEL
LIN {X 0,Y 351.275,Z 585.661,A -85,B 0,C 180,E1 -13787.765,E2 -13787.765} C_VEL
LIN {X 0,Y 352.831,Z 574.485,A -85,B 0,C 180,E1 -13789.339,E2 -13789.339} C_VEL
LIN {X 0,Y 354.356,Z 563.331,A -85,B 0,C 180,E1 -13790.612,E2 -13790.612} C_VEL
LIN {X 0,Y 355.803,Z 550.207,A -85,B 0,C 180,E1 -13791.818,E2 -13791.818} C_VEL
LIN {X 0,Y 356.552,Z 542.273,A -85,B 0,C 180,E1 -13792.418,E2 -13792.418} C_VEL
LIN {X 0,Y 354.874,Z 529.233,A -85,B 0,C 180,E1 -13793.398,E2 -13793.398} C_VEL
LIN {X 0,Y 352.408,Z 514.812,A -85,B 0,C 180,E1 -13794.276,E2 -13794.276} C_VEL
LIN {X 0,Y 347.419,Z 490.016,A -85,B 0,C 180,E1 -13795.471,E2 -13795.471} C_VEL
LIN {X 0,Y 347.905,Z 482.798,A -85,B 0,C 180,E1 -13799.001,E2 -13799.001} C_VEL
LIN {X 0,Y 348.456,Z 474.917,A -85,B 0,C 180,E1 -13802.995,E2 -13802.995} C_VEL
LIN {X 0,Y 348.878,Z 468.485,A -85,B 0,C 180,E1 -13806.314,E2 -13806.314} C_VEL
LIN {X 0,Y 349.305,Z 462.778,A -85,B 0,C 180,E1 -13809.33,E2 -13809.33} C_VEL
LIN {X 0,Y 349.896,Z 455.878,A -85,B 0,C 180,E1 -13813.073,E2 -13813.073} C_VEL
LIN {X 0,Y 350.397,Z 450.208,A -85,B 0,C 180,E1 -13816.225,E2 -13816.225} C_VEL
LIN {X 0,Y 350.417,Z 446.207,A -85,B 0,C 180,E1 -13818.559,E2 -13818.559} C_VEL
LIN {X 0,Y 349.614,Z 441.186,A -85,B 0,C 180,E1 -13821.627,E2 -13821.627} C_VEL
LIN {X 0,Y 348.502,Z 434.97,A -85,B 0,C 180,E1 -13825.622,E2 -13825.622} C_VEL
LIN {X 0,Y 347.776,Z 430.792,A -85,B 0,C 180,E1 -13828.474,E2 -13828.474} C_VEL
LIN {X 0,Y 347.806,Z 430.789,A -85,B 0,C 180,E1 -13830.99,E2 -13830.99} C_VEL
LIN {X 0,Y 347.833,Z 430.768,A -85,B 0,C 180,E1 -13833.608,E2 -13833.608} C_VEL
LIN {X 0,Y 347.79,Z 430.79,A -85,B 0,C 180,E1 -13836.162,E2 -13836.162} C_VEL
LIN {X 0,Y 347.819,Z 430.769,A -85,B 0,C 180,E1 -13839.91,E2 -13839.91} C_VEL
LIN {X 0,Y 347.868,Z 430.779,A -85,B 0,C 180,E1 -13842.359,E2 -13842.359} C_VEL
LIN {X 0,Y 347.899,Z 430.762,A -85,B 0,C 180,E1 -13845.971,E2 -13845.971} C_VEL
LIN {X 0,Y 347.898,Z 430.768,A -85,B 0,C 180,E1 -13849.525,E2 -13849.525} C_VEL
LIN {X 0,Y 348.081,Z 430.75,A -85,B 0,C 180,E1 -13853.042,E2 -13853.042} C_VEL
LIN {X 0,Y 348.208,Z 430.721,A -85,B 0,C 180,E1 -13857.687,E2 -13857.687} C_VEL
LIN {X 0,Y 348.369,Z 430.718,A -85,B 0,C 180,E1 -13860,E2 -13860} C_VEL
LIN {X 0,Y 348.208,Z 430.723,A -85,B 0,C 180,E1 -13862.314,E2 -13862.314} C_VEL
LIN {X 0,Y 348.108,Z 430.746,A -85,B 0,C 180,E1 -13866.958,E2 -13866.958} C_VEL
LIN {X 0,Y 347.969,Z 430.753,A -85,B 0,C 180,E1 -13869.299,E2 -13869.299} C_VEL
LIN {X 0,Y 347.892,Z 430.769,A -85,B 0,C 180,E1 -13872.839,E2 -13872.839} C_VEL
LIN {X 0,Y 347.841,Z 430.785,A -85,B 0,C 180,E1 -13876.431,E2 -13876.431} C_VEL
LIN {X 0,Y 347.852,Z 430.769,A -85,B 0,C 180,E1 -13878.861,E2 -13878.861} C_VEL
LIN {X 0,Y 347.765,Z 430.783,A -85,B 0,C 180,E1 -13882.58,E2 -13882.58} C_VEL
LIN {X 0,Y 347.813,Z 430.786,A -85,B 0,C 180,E1 -13885.108,E2 -13885.108} C_VEL
LIN {X 0,Y 347.812,Z 430.784,A -85,B 0,C 180,E1 -13887.694,E2 -13887.694} C_VEL
LIN {X 0,Y 347.765,Z 430.786,A -85,B 0,C 180,E1 -13890.347,E2 -13890.347} C_VEL
LIN {X 0,Y 347.746,Z 430.796,A -85,B 0,C 180,E1 -13894.464,E2 -13894.464} C_VEL
LIN {X 0,Y 347.775,Z 430.788,A -85,B 0,C 180,E1 -13897.989,E2 -13897.989} C_VEL
LIN {X 0,Y 347.749,Z 430.795,A -85,B 0,C 180,E1 -13902.025,E2 -13902.025} C_VEL
LIN {X 0,Y 347.763,Z 430.934,A -85,B 0,C 180,E1 -13902.218,E2 -13902.218} C_VEL
LIN {X 0,Y 349.404,Z 438.313,A -85,B 0,C 180,E1 -13905.251,E2 -13905.251} C_VEL
LIN {X 0,Y 350.66,Z 444.73,A -85,B 0,C 180,E1 -13907.865,E2 -13907.865} C_VEL
LIN {X 0,Y 351.521,Z 450.695,A -85,B 0,C 180,E1 -13910.225,E2 -13910.225} C_VEL
LIN {X 0,Y 351.195,Z 456.486,A -85,B 0,C 180,E1 -13912.385,E2 -13912.385} C_VEL
LIN {X 0,Y 350.608,Z 465.896,A -85,B 0,C 180,E1 -13915.857,E2 -13915.857} C_VEL
LIN {X 0,Y 349.976,Z 477.037,A -85,B 0,C 180,E1 -13919.865,E2 -13919.865} C_VEL
LIN {X 0,Y 349.355,Z 488.243,A -85,B 0,C 180,E1 -13923.732,E2 -13923.732} C_VEL
LIN {X 0,Y 349.23,Z 491.267,A -85,B 0,C 180,E1 -13924.738,E2 -13924.738} C_VEL
LIN {X 0,Y 353.646,Z 507.884,A -85,B 0,C 180,E1 -13925.57,E2 -13925.57} C_VEL
LIN {X 0,Y 356.284,Z 521.228,A -85,B 0,C 180,E1 -13926.387,E2 -13926.387} C_VEL
LIN {X 0,Y 357.681,Z 530.976,A -85,B 0,C 180,E1 -13927.09,E2 -13927.09} C_VEL
LIN {X 0,Y 356.45,Z 544.581,A -85,B 0,C 180,E1 -13928.079,E2 -13928.079} C_VEL
LIN {X 0,Y 354.976,Z 557.447,A -85,B 0,C 180,E1 -13929.274,E2 -13929.274} C_VEL
LIN {X 0,Y 353.273,Z 569.653,A -85,B 0,C 180,E1 -13930.686,E2 -13930.686} C_VEL
LIN {X 0,Y 351.751,Z 580.559,A -85,B 0,C 180,E1 -13932.26,E2 -13932.26} C_VEL
LIN {X 0,Y 350.252,Z 590.365,A -85,B 0,C 180,E1 -13933.985,E2 -13933.985} C_VEL
LIN {X 0,Y 349.322,Z 597.452,A -85,B 0,C 180,E1 -13935.475,E2 -13935.475} C_VEL
LIN {X 0,Y 348.178,Z 605.289,A -85,B 0,C 180,E1 -13937.468,E2 -13937.468} C_VEL
LIN {X 0,Y 347.305,Z 611.732,A -85,B 0,C 180,E1 -13939.507,E2 -13939.507} C_VEL
LIN {X 0,Y 346.653,Z 617.438,A -85,B 0,C 180,E1 -13941.841,E2 -13941.841} C_VEL
LIN {X 0,Y 346.338,Z 621.588,A -85,B 0,C 180,E1 -13944.177,E2 -13944.177} C_VEL
LIN {X 0,Y 346.148,Z 624.306,A -85,B 0,C 180,E1 -13946.508,E2 -13946.508} C_VEL
LIN {X 0,Y 346.058,Z 625.669,A -85,B 0,C 180,E1 -13948.836,E2 -13948.836} C_VEL
LIN {X 0,Y 346.058,Z 625.703,A -85,B 0,C 180,E1 -13951.164,E2 -13951.164} C_VEL
LIN {X 0,Y 346.146,Z 624.398,A -85,B 0,C 180,E1 -13953.492,E2 -13953.492} C_VEL
LIN {X 0,Y 346.289,Z 621.736,A -85,B 0,C 180,E1 -13955.824,E2 -13955.824} C_VEL
LIN {X 0,Y 346.652,Z 617.648,A -85,B 0,C 180,E1 -13958.159,E2 -13958.159} C_VEL
LIN {X 0,Y 347.271,Z 612.006,A -85,B 0,C 180,E1 -13960.494,E2 -13960.494} C_VEL
LIN {X 0,Y 348.146,Z 605.628,A -85,B 0,C 180,E1 -13962.533,E2 -13962.533} C_VEL
LIN {X 0,Y 349.143,Z 598.944,A -85,B 0,C 180,E1 -13964.269,E2 -13964.269} C_VEL
LIN {X 0,Y 350.245,Z 591.007,A -85,B 0,C 180,E1 -13965.986,E2 -13965.986} C_VEL
LIN {X 0,Y 351.686,Z 581.153,A -85,B 0,C 180,E1 -13967.743,E2 -13967.743} C_VEL
LIN {X 0,Y 353.18,Z 570.374,A -85,B 0,C 180,E1 -13969.319,E2 -13969.319} C_VEL
LIN {X 0,Y 354.888,Z 558.384,A -85,B 0,C 180,E1 -13970.731,E2 -13970.731} C_VEL
LIN {X 0,Y 356.332,Z 546.245,A -85,B 0,C 180,E1 -13971.883,E2 -13971.883} C_VEL
LIN {X 0,Y 357.624,Z 532.452,A -85,B 0,C 180,E1 -13972.914,E2 -13972.914} C_VEL
LIN {X 0,Y 357.16,Z 526.724,A -85,B 0,C 180,E1 -13973.329,E2 -13973.329} C_VEL
LIN {X 0,Y 354.713,Z 512.868,A -85,B 0,C 180,E1 -13974.247,E2 -13974.247} C_VEL
LIN {X 0,Y 351.264,Z 498.654,A -85,B 0,C 180,E1 -13975.017,E2 -13975.017} C_VEL
LIN {X 0,Y 349.207,Z 491.269,A -85,B 0,C 180,E1 -13975.367,E2 -13975.367} C_VEL
LIN {X 0,Y 349.732,Z 481.058,A -85,B 0,C 180,E1 -13978.835,E2 -13978.835} C_VEL
LIN {X 0,Y 350.24,Z 472.065,A -85,B 0,C 180,E1 -13982.015,E2 -13982.015} C_VEL
LIN {X 0,Y 350.338,Z 469.935,A -85,B 0,C 180,E1 -13982.785,E2 -13982.785} C_VEL
LIN {X 0,Y 349.846,Z 467.662,A -85,B 0,C 180,E1 -13983.672,E2 -13983.672} C_VEL
LIN {X 0,Y 347.287,Z 464.386,A -85,B 0,C 180,E1 -13985.151,E2 -13985.151} C_VEL
LIN {X 0,Y 345.13,Z 461.785,A -85,B 0,C 180,E1 -13986.351,E2 -13986.351} C_VEL
LIN {X 0,Y 344.307,Z 459.624,A -85,B 0,C 180,E1 -13987.263,E2 -13987.263} C_VEL
LIN {X 0,Y 344.298,Z 458.842,A -85,B 0,C 180,E1 -13987.567,E2 -13987.567} C_VEL
LIN {X 0,Y 344.688,Z 452.517,A -85,B 0,C 180,E1 -13989.96,E2 -13989.96} C_VEL
LIN {X 0,Y 343.724,Z 445.975,A -85,B 0,C 180,E1 -13992.601,E2 -13992.601} C_VEL
LIN {X 0,Y 342.122,Z 437.877,A -85,B 0,C 180,E1 -13995.971,E2 -13995.971} C_VEL
LIN {X 0,Y 340.706,Z 431.675,A -85,B 0,C 180,E1 -13998.613,E2 -13998.613} C_VEL
LIN {X 0,Y 340.735,Z 431.673,A -85,B 0,C 180,E1 -14001.773,E2 -14001.773} C_VEL
LIN {X 0,Y 340.724,Z 431.661,A -85,B 0,C 180,E1 -14005.595,E2 -14005.595} C_VEL
LIN {X 0,Y 340.706,Z 431.662,A -85,B 0,C 180,E1 -14008.956,E2 -14008.956} C_VEL
LIN {X 0,Y 340.782,Z 431.663,A -85,B 0,C 180,E1 -14012.474,E2 -14012.474} C_VEL
LIN {X 0,Y 340.799,Z 431.66,A -85,B 0,C 180,E1 -14013.55,E2 -14013.55} C_VEL
LIN {X 0,Y 345.913,Z 447.439,A -85,B 0,C 180,E1 -14014.952,E2 -14014.952} C_VEL
LIN {X 0,Y 349.919,Z 460.568,A -85,B 0,C 180,E1 -14016.316,E2 -14016.316} C_VEL
LIN {X 0,Y 348.528,Z 473.993,A -85,B 0,C 180,E1 -14017.632,E2 -14017.632} C_VEL
LIN {X 0,Y 347.018,Z 487.484,A -85,B 0,C 180,E1 -14019.242,E2 -14019.242} C_VEL
LIN {X 0,Y 345.554,Z 499.711,A -85,B 0,C 180,E1 -14021.009,E2 -14021.009} C_VEL
LIN {X 0,Y 344.235,Z 509.999,A -85,B 0,C 180,E1 -14022.78,E2 -14022.78} C_VEL
LIN {X 0,Y 342.985,Z 520.048,A -85,B 0,C 180,E1 -14024.855,E2 -14024.855} C_VEL
LIN {X 0,Y 342.18,Z 527.332,A -85,B 0,C 180,E1 -14026.64,E2 -14026.64} C_VEL
LIN {X 0,Y 341.35,Z 534.428,A -85,B 0,C 180,E1 -14028.72,E2 -14028.72} C_VEL
LIN {X 0,Y 340.706,Z 541.004,A -85,B 0,C 180,E1 -14031.1,E2 -14031.1} C_VEL
LIN {X 0,Y 340.237,Z 546.093,A -85,B 0,C 180,E1 -14033.476,E2 -14033.476} C_VEL
LIN {X 0,Y 340.181,Z 548.98,A -85,B 0,C 180,E1 -14035.26,E2 -14035.26} C_VEL
LIN {X 0,Y 340.122,Z 550.525,A -85,B 0,C 180,E1 -14036.446,E2 -14036.446} C_VEL
LIN {X 0,Y 339.749,Z 552.725,A -85,B 0,C 180,E1 -14038.815,E2 -14038.815} C_VEL
LIN {X 0,Y 339.785,Z 553.698,A -85,B 0,C 180,E1 -14041.185,E2 -14041.185} C_VEL
LIN {X 0,Y 340.173,Z 553.448,A -85,B 0,C 180,E1 -14043.553,E2 -14043.553} C_VEL
LIN {X 0,Y 340.832,Z 551.97,A -85,B 0,C 180,E1 -14045.918,E2 -14045.918} C_VEL
LIN {X 0,Y 341.444,Z 549.296,A -85,B 0,C 180,E1 -14048.284,E2 -14048.284} C_VEL
LIN {X 0,Y 342.389,Z 545.342,A -85,B 0,C 180,E1 -14050.646,E2 -14050.646} C_VEL
LIN {X 0,Y 343.447,Z 540.043,A -85,B 0,C 180,E1 -14053.008,E2 -14053.008} C_VEL
LIN {X 0,Y 345.082,Z 533.159,A -85,B 0,C 180,E1 -14055.353,E2 -14055.353} C_VEL
LIN {X 0,Y 346.357,Z 527.438,A -85,B 0,C 180,E1 -14056.954,E2 -14056.954} C_VEL
LIN {X 0,Y 348.125,Z 519.436,A -85,B 0,C 180,E1 -14058.845,E2 -14058.845} C_VEL
LIN {X 0,Y 350.239,Z 509.167,A -85,B 0,C 180,E1 -14060.866,E2 -14060.866} C_VEL
LIN {X 0,Y 352.362,Z 498.571,A -85,B 0,C 180,E1 -14062.578,E2 -14062.578} C_VEL
LIN {X 0,Y 354.713,Z 486.546,A -85,B 0,C 180,E1 -14064.187,E2 -14064.187} C_VEL
LIN {X 0,Y 356.858,Z 473.201,A -85,B 0,C 180,E1 -14065.675,E2 -14065.675} C_VEL
LIN {X 0,Y 357.607,Z 468.171,A -85,B 0,C 180,E1 -14066.161,E2 -14066.161} C_VEL
LIN {X 0,Y 355.08,Z 459.704,A -85,B 0,C 180,E1 -14067.446,E2 -14067.446} C_VEL
LIN {X 0,Y 351.325,Z 450.652,A -85,B 0,C 180,E1 -14068.955,E2 -14068.955} C_VEL
LIN {X 0,Y 347.923,Z 444.135,A -85,B 0,C 180,E1 -14070.162,E2 -14070.162} C_VEL
LIN {X 0,Y 346.272,Z 440.868,A -85,B 0,C 180,E1 -14070.778,E2 -14070.778} C_VEL
LIN {X 0,Y 344.978,Z 439.361,A -85,B 0,C 180,E1 -14071.17,E2 -14071.17} C_VEL
LIN {X 0,Y 343.248,Z 436.265,A -85,B 0,C 180,E1 -14071.797,E2 -14071.797} C_VEL
LIN {X 0,Y 341.198,Z 433.569,A -85,B 0,C 180,E1 -14072.492,E2 -14072.492} C_VEL
LIN {X 0,Y 340.678,Z 431.676,A -85,B 0,C 180,E1 -14072.8,E2 -14072.8} C_VEL
LIN {X 0,Y 340.729,Z 431.756,A -85,B 0,C 180,E1 -14075.583,E2 -14075.583} C_VEL
LIN {X 0,Y 341.281,Z 434.581,A -85,B 0,C 180,E1 -14078.507,E2 -14078.507} C_VEL
LIN {X 0,Y 342.018,Z 439.136,A -85,B 0,C 180,E1 -14082.29,E2 -14082.29} C_VEL
LIN {X 0,Y 342.099,Z 442.031,A -85,B 0,C 180,E1 -14084.306,E2 -14084.306} C_VEL
LIN {X 0,Y 341.221,Z 449.494,A -85,B 0,C 180,E1 -14088.769,E2 -14088.769} C_VEL
LIN {X 0,Y 340.854,Z 456.482,A -85,B 0,C 180,E1 -14092.537,E2 -14092.537} C_VEL
LIN {X 0,Y 340.631,Z 462.584,A -85,B 0,C 180,E1 -14095.618,E2 -14095.618} C_VEL
LIN {X 0,Y 340.365,Z 469.432,A -85,B 0,C 180,E1 -14098.922,E2 -14098.922} C_VEL
LIN {X 0,Y 340.356,Z 470.542,A -85,B 0,C 180,E1 -14099.351,E2 -14099.351} C_VEL
LIN {X 0,Y 341.201,Z 474.361,A -85,B 0,C 180,E1 -14099.77,E2 -14099.77} C_VEL
LIN {X 0,Y 342.469,Z 477.338,A -85,B 0,C 180,E1 -14100.205,E2 -14100.205} C_VEL
LIN {X 0,Y 343.612,Z 481.552,A -85,B 0,C 180,E1 -14100.685,E2 -14100.685} C_VEL
LIN {X 0,Y 346.453,Z 492.643,A -85,B 0,C 180,E1 -14101.937,E2 -14101.937} C_VEL
LIN {X 0,Y 348.876,Z 507.388,A -85,B 0,C 180,E1 -14103.448,E2 -14103.448} C_VEL
LIN {X 0,Y 349.7,Z 520.529,A -85,B 0,C 180,E1 -14104.739,E2 -14104.739} C_VEL
LIN {X 0,Y 349.521,Z 535.499,A -85,B 0,C 180,E1 -14106.287,E2 -14106.287} C_VEL
LIN {X 0,Y 349.848,Z 543.883,A -85,B 0,C 180,E1 -14107.25,E2 -14107.25} C_VEL
LIN {X 0,Y 348.576,Z 555.978,A -85,B 0,C 180,E1 -14108.248,E2 -14108.248} C_VEL
LIN {X 0,Y 347.015,Z 568.567,A -85,B 0,C 180,E1 -14109.552,E2 -14109.552} C_VEL
LIN {X 0,Y 345.407,Z 579.861,A -85,B 0,C 180,E1 -14111.001,E2 -14111.001} C_VEL
LIN {X 0,Y 343.785,Z 590.885,A -85,B 0,C 180,E1 -14112.757,E2 -14112.757} C_VEL
LIN {X 0,Y 342.449,Z 599.958,A -85,B 0,C 180,E1 -14114.526,E2 -14114.526} C_VEL
LIN {X 0,Y 341.315,Z 608.61,A -85,B 0,C 180,E1 -14116.606,E2 -14116.606} C_VEL
LIN {X 0,Y 340.267,Z 615.576,A -85,B 0,C 180,E1 -14118.684,E2 -14118.684} C_VEL
LIN {X 0,Y 339.759,Z 620.388,A -85,B 0,C 180,E1 -14120.475,E2 -14120.475} C_VEL
LIN {X 0,Y 339.339,Z 625.343,A -85,B 0,C 180,E1 -14122.862,E2 -14122.862} C_VEL
LIN {X 0,Y 339.143,Z 628.788,A -85,B 0,C 180,E1 -14125.245,E2 -14125.245} C_VEL
LIN {X 0,Y 339.051,Z 630.826,A -85,B 0,C 180,E1 -14127.624,E2 -14127.624} C_VEL
LIN {X 0,Y 339.049,Z 631.504,A -85,B 0,C 180,E1 -14130,E2 -14130} C_VEL
LIN {X 0,Y 339.051,Z 630.823,A -85,B 0,C 180,E1 -14132.376,E2 -14132.376} C_VEL
LIN {X 0,Y 339.125,Z 628.783,A -85,B 0,C 180,E1 -14134.755,E2 -14134.755} C_VEL
LIN {X 0,Y 339.318,Z 625.333,A -85,B 0,C 180,E1 -14137.139,E2 -14137.139} C_VEL
LIN {X 0,Y 339.736,Z 620.369,A -85,B 0,C 180,E1 -14139.526,E2 -14139.526} C_VEL
LIN {X 0,Y 340.262,Z 615.552,A -85,B 0,C 180,E1 -14141.316,E2 -14141.316} C_VEL
LIN {X 0,Y 341.281,Z 608.582,A -85,B 0,C 180,E1 -14143.395,E2 -14143.395} C_VEL
LIN {X 0,Y 342.395,Z 599.921,A -85,B 0,C 180,E1 -14145.476,E2 -14145.476} C_VEL
LIN {X 0,Y 343.744,Z 590.841,A -85,B 0,C 180,E1 -14147.245,E2 -14147.245} C_VEL
LIN {X 0,Y 345.061,Z 581.771,A -85,B 0,C 180,E1 -14148.711,E2 -14148.711} C_VEL
LIN {X 0,Y 346.68,Z 570.925,A -85,B 0,C 180,E1 -14150.159,E2 -14150.159} C_VEL
LIN {X 0,Y 348.25,Z 558.951,A -85,B 0,C 180,E1 -14151.463,E2 -14151.463} C_VEL
LIN {X 0,Y 349.468,Z 547.578,A -85,B 0,C 180,E1 -14152.464,E2 -14152.464} C_VEL
LIN {X 0,Y 349.801,Z 542.592,A -85,B 0,C 180,E1 -14152.846,E2 -14152.846} C_VEL
LIN {X 0,Y 348.273,Z 530.283,A -85,B 0,C 180,E1 -14153.803,E2 -14153.803} C_VEL
LIN {X 0,Y 345.881,Z 516.017,A -85,B 0,C 180,E1 -14154.711,E2 -14154.711} C_VEL
LIN {X 0,Y 342.904,Z 501.378,A -85,B 0,C 180,E1 -14155.423,E2 -14155.423} C_VEL
LIN {X 0,Y 340.417,Z 489.566,A -85,B 0,C 180,E1 -14155.937,E2 -14155.937} C_VEL
LIN {X 0,Y 340.394,Z 489.033,A -85,B 0,C 180,E1 -14156.024,E2 -14156.024} C_VEL
LIN {X 0,Y 340.952,Z 481.186,A -85,B 0,C 180,E1 -14160.033,E2 -14160.033} C_VEL
LIN {X 0,Y 341.475,Z 474.001,A -85,B 0,C 180,E1 -14163.759,E2 -14163.759} C_VEL
LIN {X 0,Y 341.977,Z 467.287,A -85,B 0,C 180,E1 -14167.323,E2 -14167.323} C_VEL
LIN {X 0,Y 342.496,Z 460.443,A -85,B 0,C 180,E1 -14171.044,E2 -14171.044} C_VEL
LIN {X 0,Y 343.175,Z 453.457,A -85,B 0,C 180,E1 -14174.953,E2 -14174.953} C_VEL
LIN {X 0,Y 343.478,Z 448.993,A -85,B 0,C 180,E1 -14177.529,E2 -14177.529} C_VEL
LIN {X 0,Y 343.097,Z 445.069,A -85,B 0,C 180,E1 -14179.91,E2 -14179.91} C_VEL
LIN {X 0,Y 342.086,Z 439.547,A -85,B 0,C 180,E1 -14183.431,E2 -14183.431} C_VEL
LIN {X 0,Y 341.183,Z 434.341,A -85,B 0,C 180,E1 -14186.916,E2 -14186.916} C_VEL
LIN {X 0,Y 340.759,Z 431.666,A -85,B 0,C 180,E1 -14188.789,E2 -14188.789} C_VEL
LIN {X 0,Y 340.78,Z 431.657,A -85,B 0,C 180,E1 -14192.474,E2 -14192.474} C_VEL
LIN {X 0,Y 340.757,Z 431.661,A -85,B 0,C 180,E1 -14195.639,E2 -14195.639} C_VEL
LIN {X 0,Y 340.749,Z 431.648,A -85,B 0,C 180,E1 -14199.474,E2 -14199.474} C_VEL
LIN {X 0,Y 340.86,Z 431.653,A -85,B 0,C 180,E1 -14201.984,E2 -14201.984} C_VEL
LIN {X 0,Y 340.871,Z 431.634,A -85,B 0,C 180,E1 -14205.705,E2 -14205.705} C_VEL
LIN {X 0,Y 340.85,Z 431.648,A -85,B 0,C 180,E1 -14209.306,E2 -14209.306} C_VEL
LIN {X 0,Y 341.049,Z 431.624,A -85,B 0,C 180,E1 -14212.898,E2 -14212.898} C_VEL
LIN {X 0,Y 341.17,Z 431.597,A -85,B 0,C 180,E1 -14217.639,E2 -14217.639} C_VEL
LIN {X 0,Y 341.318,Z 431.597,A -85,B 0,C 180,E1 -14220,E2 -14220} C_VEL
LIN {X 0,Y 341.169,Z 431.598,A -85,B 0,C 180,E1 -14222.361,E2 -14222.361} C_VEL
LIN {X 0,Y 341.078,Z 431.619,A -85,B 0,C 180,E1 -14227.102,E2 -14227.102} C_VEL
LIN {X 0,Y 340.873,Z 431.65,A -85,B 0,C 180,E1 -14230.694,E2 -14230.694} C_VEL
LIN {X 0,Y 340.865,Z 431.639,A -85,B 0,C 180,E1 -14234.325,E2 -14234.325} C_VEL
LIN {X 0,Y 340.838,Z 431.643,A -85,B 0,C 180,E1 -14238.466,E2 -14238.466} C_VEL
LIN {X 0,Y 340.719,Z 431.667,A -85,B 0,C 180,E1 -14241.842,E2 -14241.842} C_VEL
LIN {X 0,Y 340.774,Z 431.659,A -85,B 0,C 180,E1 -14245.664,E2 -14245.664} C_VEL
LIN {X 0,Y 340.743,Z 431.667,A -85,B 0,C 180,E1 -14248.32,E2 -14248.32} C_VEL
LIN {X 0,Y 340.705,Z 431.67,A -85,B 0,C 180,E1 -14251.044,E2 -14251.044} C_VEL
LIN {X 0,Y 340.719,Z 431.666,A -85,B 0,C 180,E1 -14255.279,E2 -14255.279} C_VEL
LIN {X 0,Y 340.711,Z 431.67,A -85,B 0,C 180,E1 -14258.386,E2 -14258.386} C_VEL
LIN {X 0,Y 340.752,Z 431.817,A -85,B 0,C 180,E1 -14261.613,E2 -14261.613} C_VEL
LIN {X 0,Y 342.558,Z 440.045,A -85,B 0,C 180,E1 -14265.057,E2 -14265.057} C_VEL
LIN {X 0,Y 344.018,Z 447.682,A -85,B 0,C 180,E1 -14268.216,E2 -14268.216} C_VEL
LIN {X 0,Y 344.655,Z 452.201,A -85,B 0,C 180,E1 -14270.035,E2 -14270.035} C_VEL
LIN {X 0,Y 344.526,Z 456.083,A -85,B 0,C 180,E1 -14271.525,E2 -14271.525} C_VEL
LIN {X 0,Y 343.702,Z 467.516,A -85,B 0,C 180,E1 -14275.784,E2 -14275.784} C_VEL
LIN {X 0,Y 343.134,Z 477.286,A -85,B 0,C 180,E1 -14279.343,E2 -14279.343} C_VEL
LIN {X 0,Y 342.469,Z 488.215,A -85,B 0,C 180,E1 -14283.162,E2 -14283.162} C_VEL
LIN {X 0,Y 342.348,Z 491.474,A -85,B 0,C 180,E1 -14284.212,E2 -14284.212} C_VEL
LIN {X 0,Y 346.549,Z 506.93,A -85,B 0,C 180,E1 -14284.999,E2 -14284.999} C_VEL
LIN {X 0,Y 349.426,Z 520.9,A -85,B 0,C 180,E1 -14285.875,E2 -14285.875} C_VEL
LIN {X 0,Y 351.031,Z 532.102,A -85,B 0,C 180,E1 -14286.708,E2 -14286.708} C_VEL
LIN {X 0,Y 349.774,Z 545.475,A -85,B 0,C 180,E1 -14287.715,E2 -14287.715} C_VEL
LIN {X 0,Y 348.336,Z 557.495,A -85,B 0,C 180,E1 -14288.86,E2 -14288.86} C_VEL
LIN {X 0,Y 346.727,Z 568.567,A -85,B 0,C 180,E1 -14290.153,E2 -14290.153} C_VEL
LIN {X 0,Y 345.244,Z 578.776,A -85,B 0,C 180,E1 -14291.607,E2 -14291.607} C_VEL
LIN {X 0,Y 343.671,Z 588.945,A -85,B 0,C 180,E1 -14293.364,E2 -14293.364} C_VEL
LIN {X 0,Y 342.376,Z 597.457,A -85,B 0,C 180,E1 -14295.161,E2 -14295.161} C_VEL
LIN {X 0,Y 341.417,Z 604.307,A -85,B 0,C 180,E1 -14296.913,E2 -14296.913} C_VEL
LIN {X 0,Y 340.518,Z 610.086,A -85,B 0,C 180,E1 -14298.693,E2 -14298.693} C_VEL
LIN {X 0,Y 339.751,Z 616.251,A -85,B 0,C 180,E1 -14301.075,E2 -14301.075} C_VEL
LIN {X 0,Y 339.4,Z 619.758,A -85,B 0,C 180,E1 -14302.863,E2 -14302.863} C_VEL
LIN {X 0,Y 339.133,Z 623.179,A -85,B 0,C 180,E1 -14305.245,E2 -14305.245} C_VEL
LIN {X 0,Y 338.993,Z 625.212,A -85,B 0,C 180,E1 -14307.624,E2 -14307.624} C_VEL
LIN {X 0,Y 338.978,Z 625.911,A -85,B 0,C 180,E1 -14310,E2 -14310} C_VEL
LIN {X 0,Y 338.992,Z 625.277,A -85,B 0,C 180,E1 -14312.376,E2 -14312.376} C_VEL
LIN {X 0,Y 339.123,Z 623.297,A -85,B 0,C 180,E1 -14314.755,E2 -14314.755} C_VEL
LIN {X 0,Y 339.392,Z 619.934,A -85,B 0,C 180,E1 -14317.137,E2 -14317.137} C_VEL
LIN {X 0,Y 339.899,Z 615.087,A -85,B 0,C 180,E1 -14319.521,E2 -14319.521} C_VEL
LIN {X 0,Y 340.458,Z 610.39,A -85,B 0,C 180,E1 -14321.309,E2 -14321.309} C_VEL
LIN {X 0,Y 341.542,Z 603.578,A -85,B 0,C 180,E1 -14323.385,E2 -14323.385} C_VEL
LIN {X 0,Y 342.762,Z 595.004,A -85,B 0,C 180,E1 -14325.487,E2 -14325.487} C_VEL
LIN {X 0,Y 344.088,Z 586.288,A -85,B 0,C 180,E1 -14327.227,E2 -14327.227} C_VEL
LIN {X 0,Y 345.763,Z 575.589,A -85,B 0,C 180,E1 -14328.979,E2 -14328.979} C_VEL
LIN {X 0,Y 347.364,Z 564.739,A -85,B 0,C 180,E1 -14330.427,E2 -14330.427} C_VEL
LIN {X 0,Y 348.935,Z 553.277,A -85,B 0,C 180,E1 -14331.674,E2 -14331.674} C_VEL
LIN {X 0,Y 350.319,Z 540.781,A -85,B 0,C 180,E1 -14332.772,E2 -14332.772} C_VEL
LIN {X 0,Y 351.022,Z 531.383,A -85,B 0,C 180,E1 -14333.449,E2 -14333.449} C_VEL
LIN {X 0,Y 348.875,Z 517.698,A -85,B 0,C 180,E1 -14334.445,E2 -14334.445} C_VEL
LIN {X 0,Y 345.748,Z 503.479,A -85,B 0,C 180,E1 -14335.299,E2 -14335.299} C_VEL
LIN {X 0,Y 342.321,Z 491.251,A -85,B 0,C 180,E1 -14335.92,E2 -14335.92} C_VEL
LIN {X 0,Y 342.89,Z 480.953,A -85,B 0,C 180,E1 -14339.466,E2 -14339.466} C_VEL
LIN {X 0,Y 343.456,Z 471.22,A -85,B 0,C 180,E1 -14342.968,E2 -14342.968} C_VEL
LIN {X 0,Y 344.054,Z 462.145,A -85,B 0,C 180,E1 -14346.326,E2 -14346.326} C_VEL
LIN {X 0,Y 344.298,Z 458.842,A -85,B 0,C 180,E1 -14347.567,E2 -14347.567} C_VEL
LIN {X 0,Y 343.827,Z 456.651,A -85,B 0,C 180,E1 -14348.474,E2 -14348.474} C_VEL
LIN {X 0,Y 342.38,Z 454.721,A -85,B 0,C 180,E1 -14349.382,E2 -14349.382} C_VEL
LIN {X 0,Y 337.613,Z 449.851,A -85,B 0,C 180,E1 -14351.833,E2 -14351.833} C_VEL
LIN {X 0,Y 337.024,Z 448.414,A -85,B 0,C 180,E1 -14352.464,E2 -14352.464} C_VEL
LIN {X 0,Y 335.255,Z 439.564,A -85,B 0,C 180,E1 -14356.228,E2 -14356.228} C_VEL
LIN {X 0,Y 333.629,Z 432.562,A -85,B 0,C 180,E1 -14359.319,E2 -14359.319} C_VEL
LIN {X 0,Y 333.667,Z 432.543,A -85,B 0,C 180,E1 -14363.168,E2 -14363.168} C_VEL
LIN {X 0,Y 333.676,Z 432.54,A -85,B 0,C 180,E1 -14365.341,E2 -14365.341} C_VEL
LIN {X 0,Y 333.704,Z 432.53,A -85,B 0,C 180,E1 -14369.71,E2 -14369.71} C_VEL
LIN {X 0,Y 333.78,Z 432.585,A -85,B 0,C 180,E1 -14373.172,E2 -14373.172} C_VEL
LIN {X 0,Y 338.621,Z 447.55,A -85,B 0,C 180,E1 -14374.532,E2 -14374.532} C_VEL
LIN {X 0,Y 342.781,Z 461.005,A -85,B 0,C 180,E1 -14375.952,E2 -14375.952} C_VEL
LIN {X 0,Y 343.023,Z 462.726,A -85,B 0,C 180,E1 -14376.131,E2 -14376.131} C_VEL
LIN {X 0,Y 341.533,Z 476.222,A -85,B 0,C 180,E1 -14377.512,E2 -14377.512} C_VEL
LIN {X 0,Y 340.03,Z 489.118,A -85,B 0,C 180,E1 -14379.112,E2 -14379.112} C_VEL
LIN {X 0,Y 338.513,Z 501.198,A -85,B 0,C 180,E1 -14380.914,E2 -14380.914} C_VEL
LIN {X 0,Y 337.178,Z 511.384,A -85,B 0,C 180,E1 -14382.721,E2 -14382.721} C_VEL
LIN {X 0,Y 336.04,Z 520.071,A -85,B 0,C 180,E1 -14384.534,E2 -14384.534} C_VEL
LIN {X 0,Y 335.22,Z 527.436,A -85,B 0,C 180,E1 -14386.358,E2 -14386.358} C_VEL
LIN {X 0,Y 334.352,Z 534.674,A -85,B 0,C 180,E1 -14388.481,E2 -14388.481} C_VEL
LIN {X 0,Y 333.685,Z 541.379,A -85,B 0,C 180,E1 -14390.911,E2 -14390.911} C_VEL
LIN {X 0,Y 333.202,Z 546.586,A -85,B 0,C 180,E1 -14393.338,E2 -14393.338} C_VEL
LIN {X 0,Y 333.134,Z 549.579,A -85,B 0,C 180,E1 -14395.159,E2 -14395.159} C_VEL
LIN {X 0,Y 333.088,Z 551.173,A -85,B 0,C 180,E1 -14396.371,E2 -14396.371} C_VEL
LIN {X 0,Y 332.706,Z 553.469,A -85,B 0,C 180,E1 -14398.79,E2 -14398.79} C_VEL
LIN {X 0,Y 332.74,Z 554.535,A -85,B 0,C 180,E1 -14401.21,E2 -14401.21} C_VEL
LIN {X 0,Y 333.149,Z 554.358,A -85,B 0,C 180,E1 -14403.628,E2 -14403.628} C_VEL
LIN {X 0,Y 333.839,Z 552.961,A -85,B 0,C 180,E1 -14406.042,E2 -14406.042} C_VEL
LIN {X 0,Y 334.503,Z 550.405,A -85,B 0,C 180,E1 -14408.457,E2 -14408.457} C_VEL
LIN {X 0,Y 335.505,Z 546.561,A -85,B 0,C 180,E1 -14410.867,E2 -14410.867} C_VEL
LIN {X 0,Y 336.674,Z 541.366,A -85,B 0,C 180,E1 -14413.275,E2 -14413.275} C_VEL
LIN {X 0,Y 338.391,Z 534.656,A -85,B 0,C 180,E1 -14415.664,E2 -14415.664} C_VEL
LIN {X 0,Y 339.917,Z 528.446,A -85,B 0,C 180,E1 -14417.445,E2 -14417.445} C_VEL
LIN {X 0,Y 341.963,Z 519.901,A -85,B 0,C 180,E1 -14419.51,E2 -14419.51} C_VEL
LIN {X 0,Y 344.232,Z 509.554,A -85,B 0,C 180,E1 -14421.561,E2 -14421.561} C_VEL
LIN {X 0,Y 346.532,Z 498.992,A -85,B 0,C 180,E1 -14423.296,E2 -14423.296} C_VEL
LIN {X 0,Y 348.978,Z 487.251,A -85,B 0,C 180,E1 -14424.876,E2 -14424.876} C_VEL
LIN {X 0,Y 351.132,Z 474.908,A -85,B 0,C 180,E1 -14426.295,E2 -14426.295} C_VEL
LIN {X 0,Y 351.69,Z 470.468,A -85,B 0,C 180,E1 -14426.759,E2 -14426.759} C_VEL
LIN {X 0,Y 349.114,Z 461.898,A -85,B 0,C 180,E1 -14428.17,E2 -14428.17} C_VEL
LIN {X 0,Y 345.931,Z 453.97,A -85,B 0,C 180,E1 -14429.589,E2 -14429.589} C_VEL
LIN {X 0,Y 341.508,Z 445.535,A -85,B 0,C 180,E1 -14431.323,E2 -14431.323} C_VEL
LIN {X 0,Y 338.772,Z 441.11,A -85,B 0,C 180,E1 -14432.385,E2 -14432.385} C_VEL
LIN {X 0,Y 337.748,Z 439.794,A -85,B 0,C 180,E1 -14432.753,E2 -14432.753} C_VEL
LIN {X 0,Y 336.323,Z 437.259,A -85,B 0,C 180,E1 -14433.383,E2 -14433.383} C_VEL
LIN {X 0,Y 334.364,Z 434.839,A -85,B 0,C 180,E1 -14434.141,E2 -14434.141} C_VEL
LIN {X 0,Y 333.703,Z 432.611,A -85,B 0,C 180,E1 -14434.588,E2 -14434.588} C_VEL
LIN {X 0,Y 334.16,Z 435.267,A -85,B 0,C 180,E1 -14437.584,E2 -14437.584} C_VEL
LIN {X 0,Y 334.823,Z 438.911,A -85,B 0,C 180,E1 -14440.918,E2 -14440.918} C_VEL
LIN {X 0,Y 335.139,Z 441.282,A -85,B 0,C 180,E1 -14442.78,E2 -14442.78} C_VEL
LIN {X 0,Y 335.09,Z 443.765,A -85,B 0,C 180,E1 -14444.512,E2 -14444.512} C_VEL
LIN {X 0,Y 334.169,Z 451.479,A -85,B 0,C 180,E1 -14449.211,E2 -14449.211} C_VEL
LIN {X 0,Y 333.785,Z 458.636,A -85,B 0,C 180,E1 -14453.14,E2 -14453.14} C_VEL
LIN {X 0,Y 333.534,Z 464.3,A -85,B 0,C 180,E1 -14456.055,E2 -14456.055} C_VEL
LIN {X 0,Y 333.438,Z 467.717,A -85,B 0,C 180,E1 -14457.701,E2 -14457.701} C_VEL
LIN {X 0,Y 334.357,Z 471.914,A -85,B 0,C 180,E1 -14458.241,E2 -14458.241} C_VEL
LIN {X 0,Y 335.739,Z 475.272,A -85,B 0,C 180,E1 -14458.796,E2 -14458.796} C_VEL
LIN {X 0,Y 336.906,Z 479.474,A -85,B 0,C 180,E1 -14459.346,E2 -14459.346} C_VEL
LIN {X 0,Y 339.265,Z 488.096,A -85,B 0,C 180,E1 -14460.464,E2 -14460.464} C_VEL
LIN {X 0,Y 341.227,Z 497.164,A -85,B 0,C 180,E1 -14461.54,E2 -14461.54} C_VEL
LIN {X 0,Y 342.983,Z 509.719,A -85,B 0,C 180,E1 -14462.917,E2 -14462.917} C_VEL
LIN {X 0,Y 343.54,Z 521.647,A -85,B 0,C 180,E1 -14464.176,E2 -14464.176} C_VEL
LIN {X 0,Y 343.108,Z 536.693,A -85,B 0,C 180,E1 -14465.816,E2 -14465.816} C_VEL
LIN {X 0,Y 343.148,Z 545.844,A -85,B 0,C 180,E1 -14466.94,E2 -14466.94} C_VEL
LIN {X 0,Y 341.593,Z 559.111,A -85,B 0,C 180,E1 -14468.11,E2 -14468.11} C_VEL
LIN {X 0,Y 340.005,Z 570.948,A -85,B 0,C 180,E1 -14469.427,E2 -14469.427} C_VEL
LIN {X 0,Y 338.36,Z 581.778,A -85,B 0,C 180,E1 -14470.905,E2 -14470.905} C_VEL
LIN {X 0,Y 336.693,Z 592.459,A -85,B 0,C 180,E1 -14472.696,E2 -14472.696} C_VEL
LIN {X 0,Y 335.277,Z 601.835,A -85,B 0,C 180,E1 -14474.632,E2 -14474.632} C_VEL
LIN {X 0,Y 334.213,Z 609.671,A -85,B 0,C 180,E1 -14476.626,E2 -14476.626} C_VEL
LIN {X 0,Y 333.268,Z 615.52,A -85,B 0,C 180,E1 -14478.443,E2 -14478.443} C_VEL
LIN {X 0,Y 332.728,Z 620.332,A -85,B 0,C 180,E1 -14480.272,E2 -14480.272} C_VEL
LIN {X 0,Y 332.267,Z 625.286,A -85,B 0,C 180,E1 -14482.709,E2 -14482.709} C_VEL
LIN {X 0,Y 332.048,Z 628.73,A -85,B 0,C 180,E1 -14485.143,E2 -14485.143} C_VEL
LIN {X 0,Y 331.966,Z 630.768,A -85,B 0,C 180,E1 -14487.573,E2 -14487.573} C_VEL
LIN {X 0,Y 331.952,Z 631.445,A -85,B 0,C 180,E1 -14490,E2 -14490} C_VEL
LIN {X 0,Y 331.965,Z 630.765,A -85,B 0,C 180,E1 -14492.427,E2 -14492.427} C_VEL
LIN {X 0,Y 332.029,Z 628.724,A -85,B 0,C 180,E1 -14494.857,E2 -14494.857} C_VEL
LIN {X 0,Y 332.254,Z 625.275,A -85,B 0,C 180,E1 -14497.291,E2 -14497.291} C_VEL
LIN {X 0,Y 332.71,Z 620.311,A -85,B 0,C 180,E1 -14499.729,E2 -14499.729} C_VEL
LIN {X 0,Y 333.53,Z 613.687,A -85,B 0,C 180,E1 -14502.164,E2 -14502.164} C_VEL
LIN {X 0,Y 334.577,Z 606.269,A -85,B 0,C 180,E1 -14504.289,E2 -14504.289} C_VEL
LIN {X 0,Y 335.755,Z 598.5,A -85,B 0,C 180,E1 -14506.102,E2 -14506.102} C_VEL
LIN {X 0,Y 337.203,Z 589.109,A -85,B 0,C 180,E1 -14507.904,E2 -14507.904} C_VEL
LIN {X 0,Y 338.788,Z 578.685,A -85,B 0,C 180,E1 -14509.543,E2 -14509.543} C_VEL
LIN {X 0,Y 340.505,Z 567.158,A -85,B 0,C 180,E1 -14511.015,E2 -14511.015} C_VEL
LIN {X 0,Y 341.937,Z 555.85,A -85,B 0,C 180,E1 -14512.196,E2 -14512.196} C_VEL
LIN {X 0,Y 343.164,Z 544.405,A -85,B 0,C 180,E1 -14513.164,E2 -14513.164} C_VEL
LIN {X 0,Y 341.661,Z 531.31,A -85,B 0,C 180,E1 -14514.227,E2 -14514.227} C_VEL
LIN {X 0,Y 339.311,Z 516.752,A -85,B 0,C 180,E1 -14515.189,E2 -14515.189} C_VEL
LIN {X 0,Y 336.355,Z 501.961,A -85,B 0,C 180,E1 -14515.94,E2 -14515.94} C_VEL
LIN {X 0,Y 333.486,Z 489.549,A -85,B 0,C 180,E1 -14516.477,E2 -14516.477} C_VEL
LIN {X 0,Y 333.392,Z 487.98,A -85,B 0,C 180,E1 -14516.697,E2 -14516.697} C_VEL
LIN {X 0,Y 333.906,Z 480.974,A -85,B 0,C 180,E1 -14520.349,E2 -14520.349} C_VEL
LIN {X 0,Y 334.415,Z 474.4,A -85,B 0,C 180,E1 -14523.843,E2 -14523.843} C_VEL
LIN {X 0,Y 334.932,Z 467.693,A -85,B 0,C 180,E1 -14527.482,E2 -14527.482} C_VEL
LIN {X 0,Y 335.428,Z 461.269,A -85,B 0,C 180,E1 -14531.037,E2 -14531.037} C_VEL
LIN {X 0,Y 336.078,Z 454.882,A -85,B 0,C 180,E1 -14534.683,E2 -14534.683} C_VEL
LIN {X 0,Y 336.399,Z 450.921,A -85,B 0,C 180,E1 -14536.988,E2 -14536.988} C_VEL
LIN {X 0,Y 336.163,Z 446.658,A -85,B 0,C 180,E1 -14539.601,E2 -14539.601} C_VEL
LIN {X 0,Y 335.244,Z 441.656,A -85,B 0,C 180,E1 -14542.809,E2 -14542.809} C_VEL
LIN {X 0,Y 334.411,Z 436.694,A -85,B 0,C 180,E1 -14546.157,E2 -14546.157} C_VEL
LIN {X 0,Y 333.701,Z 432.546,A -85,B 0,C 180,E1 -14549.112,E2 -14549.112} C_VEL
LIN {X 0,Y 333.744,Z 432.534,A -85,B 0,C 180,E1 -14552.401,E2 -14552.401} C_VEL
LIN {X 0,Y 333.728,Z 432.531,A -85,B 0,C 180,E1 -14555.091,E2 -14555.091} C_VEL
LIN {X 0,Y 333.683,Z 432.529,A -85,B 0,C 180,E1 -14559.019,E2 -14559.019} C_VEL
LIN {X 0,Y 333.796,Z 432.53,A -85,B 0,C 180,E1 -14561.59,E2 -14561.59} C_VEL
LIN {X 0,Y 333.809,Z 432.513,A -85,B 0,C 180,E1 -14565.577,E2 -14565.577} C_VEL
LIN {X 0,Y 333.819,Z 432.526,A -85,B 0,C 180,E1 -14569.078,E2 -14569.078} C_VEL
LIN {X 0,Y 333.995,Z 432.5,A -85,B 0,C 180,E1 -14572.747,E2 -14572.747} C_VEL
LIN {X 0,Y 333.811,Z 432.526,A -85,B 0,C 180,E1 -14575.169,E2 -14575.169} C_VEL
LIN {X 0,Y 334.107,Z 432.476,A -85,B 0,C 180,E1 -14577.589,E2 -14577.589} C_VEL
LIN {X 0,Y 334.268,Z 432.475,A -85,B 0,C 180,E1 -14580,E2 -14580} C_VEL
LIN {X 0,Y 334.106,Z 432.477,A -85,B 0,C 180,E1 -14582.411,E2 -14582.411} C_VEL
LIN {X 0,Y 334.027,Z 432.495,A -85,B 0,C 180,E1 -14587.253,E2 -14587.253} C_VEL
LIN {X 0,Y 333.836,Z 432.528,A -85,B 0,C 180,E1 -14590.922,E2 -14590.922} C_VEL
LIN {X 0,Y 333.81,Z 432.52,A -85,B 0,C 180,E1 -14594.634,E2 -14594.634} C_VEL
LIN {X 0,Y 333.797,Z 432.519,A -85,B 0,C 180,E1 -14598.655,E2 -14598.655} C_VEL
LIN {X 0,Y 333.658,Z 432.541,A -85,B 0,C 180,E1 -14602.281,E2 -14602.281} C_VEL
LIN {X 0,Y 333.737,Z 432.532,A -85,B 0,C 180,E1 -14606.246,E2 -14606.246} C_VEL
LIN {X 0,Y 333.712,Z 432.541,A -85,B 0,C 180,E1 -14608.972,E2 -14608.972} C_VEL
LIN {X 0,Y 333.645,Z 432.547,A -85,B 0,C 180,E1 -14612.587,E2 -14612.587} C_VEL
LIN {X 0,Y 333.678,Z 432.543,A -85,B 0,C 180,E1 -14616.139,E2 -14616.139} C_VEL
LIN {X 0,Y 333.648,Z 432.551,A -85,B 0,C 180,E1 -14619.192,E2 -14619.192} C_VEL
LIN {X 0,Y 333.66,Z 432.757,A -85,B 0,C 180,E1 -14620.965,E2 -14620.965} C_VEL
LIN {X 0,Y 335.587,Z 441.173,A -85,B 0,C 180,E1 -14624.599,E2 -14624.599} C_VEL
LIN {X 0,Y 336.945,Z 448.163,A -85,B 0,C 180,E1 -14627.551,E2 -14627.551} C_VEL
LIN {X 0,Y 337.797,Z 453.707,A -85,B 0,C 180,E1 -14629.837,E2 -14629.837} C_VEL
LIN {X 0,Y 337.513,Z 459.158,A -85,B 0,C 180,E1 -14631.923,E2 -14631.923} C_VEL
LIN {X 0,Y 336.817,Z 469.181,A -85,B 0,C 180,E1 -14635.71,E2 -14635.71} C_VEL
LIN {X 0,Y 336.185,Z 479.278,A -85,B 0,C 180,E1 -14639.424,E2 -14639.424} C_VEL
LIN {X 0,Y 335.515,Z 490.13,A -85,B 0,C 180,E1 -14643.234,E2 -14643.234} C_VEL
LIN {X 0,Y 335.49,Z 491.367,A -85,B 0,C 180,E1 -14643.644,E2 -14643.644} C_VEL
LIN {X 0,Y 339.855,Z 507.224,A -85,B 0,C 180,E1 -14644.483,E2 -14644.483} C_VEL
LIN {X 0,Y 342.708,Z 521.158,A -85,B 0,C 180,E1 -14645.384,E2 -14645.384} C_VEL
LIN {X 0,Y 344.413,Z 533.23,A -85,B 0,C 180,E1 -14646.314,E2 -14646.314} C_VEL
LIN {X 0,Y 343.118,Z 546.347,A -85,B 0,C 180,E1 -14647.336,E2 -14647.336} C_VEL
LIN {X 0,Y 341.546,Z 558.923,A -85,B 0,C 180,E1 -14648.577,E2 -14648.577} C_VEL
LIN {X 0,Y 339.685,Z 570.816,A -85,B 0,C 180,E1 -14650.039,E2 -14650.039} C_VEL
LIN {X 0,Y 338.218,Z 580.668,A -85,B 0,C 180,E1 -14651.525,E2 -14651.525} C_VEL
LIN {X 0,Y 336.574,Z 590.476,A -85,B 0,C 180,E1 -14653.315,E2 -14653.315} C_VEL
LIN {X 0,Y 335.372,Z 598.311,A -85,B 0,C 180,E1 -14655.047,E2 -14655.047} C_VEL
LIN {X 0,Y 334.305,Z 605.405,A -85,B 0,C 180,E1 -14656.939,E2 -14656.939} C_VEL
LIN {X 0,Y 333.314,Z 611.849,A -85,B 0,C 180,E1 -14659.061,E2 -14659.061} C_VEL
LIN {X 0,Y 332.564,Z 617.556,A -85,B 0,C 180,E1 -14661.493,E2 -14661.493} C_VEL
LIN {X 0,Y 332.181,Z 621.706,A -85,B 0,C 180,E1 -14663.928,E2 -14663.928} C_VEL
LIN {X 0,Y 332.004,Z 624.423,A -85,B 0,C 180,E1 -14666.359,E2 -14666.359} C_VEL
